// TIA Portal V17 export
// export: Created 2025-03-12T15:33:50.5234249Z, ExportSetting WithDefaults, DisplayName Totally Integrated Automation Portal, DisplayVersion V17 Update 8, DisplayName TIA Portal Openness, DisplayVersion V17 Update 8, DisplayName TIA Portal Version Control Interface, DisplayVersion V17, DisplayName SINAMICS Startdrive Advanced, DisplayVersion V17 SP2, DisplayName SINAMICS Startdrive G110M, G120, G120C, G120D, G120P, G115D, DisplayVersion V17 SP2, DisplayName SINAMICS Startdrive G130, G150, S120, S150, SINAMICS MV, S210, DisplayVersion V17 SP2, DisplayName STEP 7 Professional, DisplayVersion V17 Update 8, DisplayName SINUMERIK ONE STEP 7 Toolbox, DisplayVersion V17 Update 12, DisplayName SINUMERIK 840D sl STEP 7 Toolbox, DisplayVersion V17 Update 12, DisplayName STEP 7 Safety, DisplayVersion V17 Update 6, DisplayName WinCC Advanced, DisplayVersion V17 Update 8
FUNCTION "FC1101_MACHINE_SEQUENCE" : Void   // FC1101, LAD
{ S7_Optimized_Access := 'FALSE' }
AUTHOR : ETXETAR
VERSION : 1.0
// stored: AutoNumber false, IsIECCheckEnabled false, SetENOAutomatically false, UDAEnableTagReadback false
   VAR_TEMP
      PHD_ARM1 : Bool;   // PART HANDLING DEVICE ARM 1
      PHD_ARM2 : Bool;   // PART HANDLING DEVICE ARM 2
      QC_AUXILIARY : Bool;   // QUALITY CHECK AUXILIARY
   END_VAR
   VAR CONSTANT
      FC_NUMBER : DInt := 1101;   // FC NUMBER
   END_VAR
   VAR_TEMP   // added for the SCL form of the ladder/FBD networks
      _w1 : Bool;
      _w2 : Bool;
      _w3 : Bool;
   END_VAR
BEGIN

REGION Network 1: GENERAL CONDITIONS
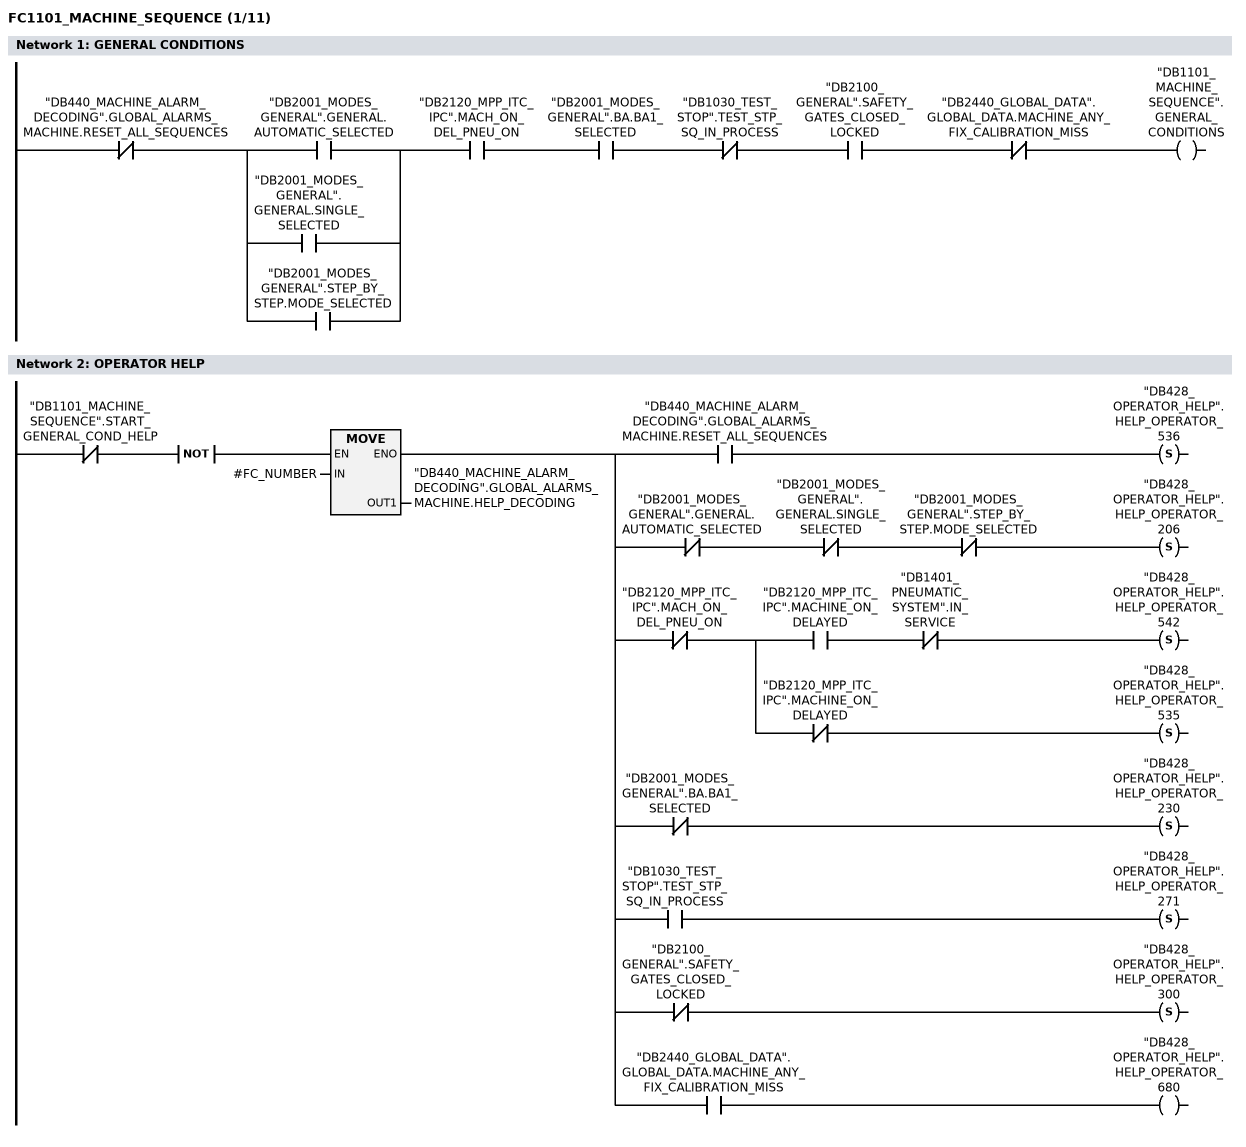
   RUNG wire#powerrail
      I_Contact( "DB440_MACHINE_ALARM_DECODING".GLOBAL_ALARMS_MACHINE.RESET_ALL_SEQUENCES )
      wire#w1
      Contact( "DB2001_MODES_GENERAL".GENERAL.AUTOMATIC_SELECTED )
      wire#w2
      Contact( "DB2120_MPP_ITC_IPC".MACH_ON_DEL_PNEU_ON )
      Contact( "DB2001_MODES_GENERAL".BA.BA1_SELECTED )
      I_Contact( "DB1030_TEST_STOP".TEST_STP_SQ_IN_PROCESS )
      Contact( "DB2100_GENERAL".SAFETY_GATES_CLOSED_LOCKED )
      I_Contact( "DB2440_GLOBAL_DATA".GLOBAL_DATA.MACHINE_ANY_FIX_CALIBRATION_MISS )
      Coil( "DB1101_MACHINE_SEQUENCE".GENERAL_CONDITIONS )
   END_RUNG
   RUNG wire#w1
      Contact( "DB2001_MODES_GENERAL".GENERAL.SINGLE_SELECTED )
   END_RUNG wire#w2
   RUNG wire#w1
      Contact( "DB2001_MODES_GENERAL".STEP_BY_STEP.MODE_SELECTED )
   END_RUNG wire#w2
   // the same network as SCL:
   "DB1101_MACHINE_SEQUENCE".GENERAL_CONDITIONS := NOT "DB440_MACHINE_ALARM_DECODING".GLOBAL_ALARMS_MACHINE.RESET_ALL_SEQUENCES AND ("DB2001_MODES_GENERAL".GENERAL.AUTOMATIC_SELECTED OR "DB2001_MODES_GENERAL".GENERAL.SINGLE_SELECTED OR "DB2001_MODES_GENERAL".STEP_BY_STEP.MODE_SELECTED) AND "DB2120_MPP_ITC_IPC".MACH_ON_DEL_PNEU_ON AND "DB2001_MODES_GENERAL".BA.BA1_SELECTED AND NOT "DB1030_TEST_STOP".TEST_STP_SQ_IN_PROCESS AND "DB2100_GENERAL".SAFETY_GATES_CLOSED_LOCKED AND NOT "DB2440_GLOBAL_DATA".GLOBAL_DATA.MACHINE_ANY_FIX_CALIBRATION_MISS;
END_REGION

REGION Network 2: OPERATOR HELP
   RUNG wire#powerrail
      I_Contact( "DB1101_MACHINE_SEQUENCE".START_GENERAL_COND_HELP )
      Not()
      { S7_GenerateENO := "TRUE" } Move(in := #FC_NUMBER, out1 => "DB440_MACHINE_ALARM_DECODING".GLOBAL_ALARMS_MACHINE.HELP_DECODING)
      wire#w1
      Contact( "DB440_MACHINE_ALARM_DECODING".GLOBAL_ALARMS_MACHINE.RESET_ALL_SEQUENCES )
      S_Coil( "DB428_OPERATOR_HELP".HELP_OPERATOR_536 )
   END_RUNG
   RUNG wire#w1
      I_Contact( "DB2001_MODES_GENERAL".GENERAL.AUTOMATIC_SELECTED )
      I_Contact( "DB2001_MODES_GENERAL".GENERAL.SINGLE_SELECTED )
      I_Contact( "DB2001_MODES_GENERAL".STEP_BY_STEP.MODE_SELECTED )
      S_Coil( "DB428_OPERATOR_HELP".HELP_OPERATOR_206 )
   END_RUNG
   RUNG wire#w1
      I_Contact( "DB2120_MPP_ITC_IPC".MACH_ON_DEL_PNEU_ON )
      wire#w2
      Contact( "DB2120_MPP_ITC_IPC".MACHINE_ON_DELAYED )
      I_Contact( "DB1401_PNEUMATIC_SYSTEM".IN_SERVICE )
      S_Coil( "DB428_OPERATOR_HELP".HELP_OPERATOR_542 )
   END_RUNG
   RUNG wire#w2
      I_Contact( "DB2120_MPP_ITC_IPC".MACHINE_ON_DELAYED )
      S_Coil( "DB428_OPERATOR_HELP".HELP_OPERATOR_535 )
   END_RUNG
   RUNG wire#w1
      I_Contact( "DB2001_MODES_GENERAL".BA.BA1_SELECTED )
      S_Coil( "DB428_OPERATOR_HELP".HELP_OPERATOR_230 )
   END_RUNG
   RUNG wire#w1
      Contact( "DB1030_TEST_STOP".TEST_STP_SQ_IN_PROCESS )
      S_Coil( "DB428_OPERATOR_HELP".HELP_OPERATOR_271 )
   END_RUNG
   RUNG wire#w1
      I_Contact( "DB2100_GENERAL".SAFETY_GATES_CLOSED_LOCKED )
      S_Coil( "DB428_OPERATOR_HELP".HELP_OPERATOR_300 )
   END_RUNG
   RUNG wire#w1
      Contact( "DB2440_GLOBAL_DATA".GLOBAL_DATA.MACHINE_ANY_FIX_CALIBRATION_MISS )
      Coil( "DB428_OPERATOR_HELP".HELP_OPERATOR_680 )
   END_RUNG
   // the same network as SCL:
   // ENO of a box is taken as its EN; it also drops when the box reports an error
   #_w1 := NOT (NOT "DB1101_MACHINE_SEQUENCE".START_GENERAL_COND_HELP);
   IF #_w1 THEN "DB440_MACHINE_ALARM_DECODING".GLOBAL_ALARMS_MACHINE.HELP_DECODING := #FC_NUMBER; END_IF;
   IF #_w1 AND "DB440_MACHINE_ALARM_DECODING".GLOBAL_ALARMS_MACHINE.RESET_ALL_SEQUENCES THEN
       "DB428_OPERATOR_HELP".HELP_OPERATOR_536 := TRUE;
   END_IF;
   IF #_w1 AND NOT "DB2001_MODES_GENERAL".GENERAL.AUTOMATIC_SELECTED AND NOT "DB2001_MODES_GENERAL".GENERAL.SINGLE_SELECTED AND NOT "DB2001_MODES_GENERAL".STEP_BY_STEP.MODE_SELECTED THEN
       "DB428_OPERATOR_HELP".HELP_OPERATOR_206 := TRUE;
   END_IF;
   #_w2 := #_w1 AND NOT "DB2120_MPP_ITC_IPC".MACH_ON_DEL_PNEU_ON;
   IF #_w2 AND "DB2120_MPP_ITC_IPC".MACHINE_ON_DELAYED AND NOT "DB1401_PNEUMATIC_SYSTEM".IN_SERVICE THEN
       "DB428_OPERATOR_HELP".HELP_OPERATOR_542 := TRUE;
   END_IF;
   IF #_w2 AND NOT "DB2120_MPP_ITC_IPC".MACHINE_ON_DELAYED THEN
       "DB428_OPERATOR_HELP".HELP_OPERATOR_535 := TRUE;
   END_IF;
   IF #_w1 AND NOT "DB2001_MODES_GENERAL".BA.BA1_SELECTED THEN
       "DB428_OPERATOR_HELP".HELP_OPERATOR_230 := TRUE;
   END_IF;
   IF #_w1 AND "DB1030_TEST_STOP".TEST_STP_SQ_IN_PROCESS THEN
       "DB428_OPERATOR_HELP".HELP_OPERATOR_271 := TRUE;
   END_IF;
   IF #_w1 AND NOT "DB2100_GENERAL".SAFETY_GATES_CLOSED_LOCKED THEN
       "DB428_OPERATOR_HELP".HELP_OPERATOR_300 := TRUE;
   END_IF;
   "DB428_OPERATOR_HELP".HELP_OPERATOR_680 := #_w1 AND "DB2440_GLOBAL_DATA".GLOBAL_DATA.MACHINE_ANY_FIX_CALIBRATION_MISS;
END_REGION

REGION Network 3: INITIAL CONDITIONS
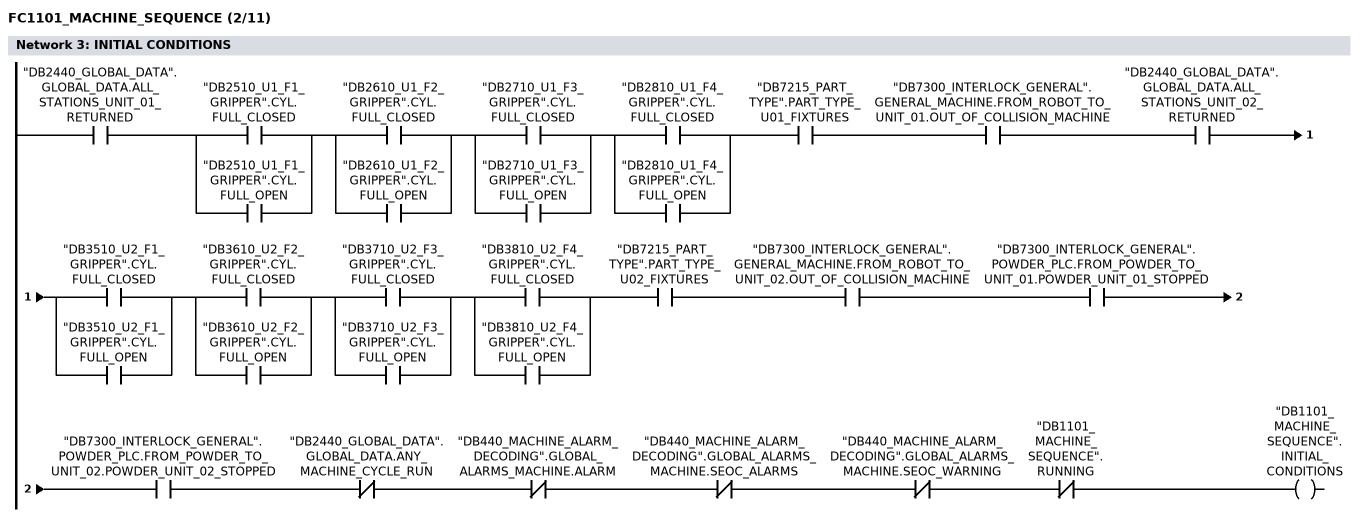
   RUNG wire#powerrail
      Contact( "DB2440_GLOBAL_DATA".GLOBAL_DATA.ALL_STATIONS_UNIT_01_RETURNED )
      wire#w1
      Contact( "DB2510_U1_F1_GRIPPER".CYL.FULL_CLOSED )
      wire#w2
      Contact( "DB2610_U1_F2_GRIPPER".CYL.FULL_CLOSED )
      wire#w3
      Contact( "DB2710_U1_F3_GRIPPER".CYL.FULL_CLOSED )
      wire#w4
      Contact( "DB2810_U1_F4_GRIPPER".CYL.FULL_CLOSED )
      wire#w5
      Contact( "DB7215_PART_TYPE".PART_TYPE_U01_FIXTURES )
      Contact( "DB7300_INTERLOCK_GENERAL".GENERAL_MACHINE.FROM_ROBOT_TO_UNIT_01.OUT_OF_COLLISION_MACHINE )
      Contact( "DB2440_GLOBAL_DATA".GLOBAL_DATA.ALL_STATIONS_UNIT_02_RETURNED )
      wire#w6
      Contact( "DB3510_U2_F1_GRIPPER".CYL.FULL_CLOSED )
      wire#w7
      Contact( "DB3610_U2_F2_GRIPPER".CYL.FULL_CLOSED )
      wire#w8
      Contact( "DB3710_U2_F3_GRIPPER".CYL.FULL_CLOSED )
      wire#w9
      Contact( "DB3810_U2_F4_GRIPPER".CYL.FULL_CLOSED )
      wire#w10
      Contact( "DB7215_PART_TYPE".PART_TYPE_U02_FIXTURES )
      Contact( "DB7300_INTERLOCK_GENERAL".GENERAL_MACHINE.FROM_ROBOT_TO_UNIT_02.OUT_OF_COLLISION_MACHINE )
      Contact( "DB7300_INTERLOCK_GENERAL".POWDER_PLC.FROM_POWDER_TO_UNIT_01.POWDER_UNIT_01_STOPPED )
      Contact( "DB7300_INTERLOCK_GENERAL".POWDER_PLC.FROM_POWDER_TO_UNIT_02.POWDER_UNIT_02_STOPPED )
      I_Contact( "DB2440_GLOBAL_DATA".GLOBAL_DATA.ANY_MACHINE_CYCLE_RUN )
      I_Contact( "DB440_MACHINE_ALARM_DECODING".GLOBAL_ALARMS_MACHINE.ALARM )
      I_Contact( "DB440_MACHINE_ALARM_DECODING".GLOBAL_ALARMS_MACHINE.SEOC_ALARMS )
      I_Contact( "DB440_MACHINE_ALARM_DECODING".GLOBAL_ALARMS_MACHINE.SEOC_WARNING )
      I_Contact( "DB1101_MACHINE_SEQUENCE".RUNNING )
      Coil( "DB1101_MACHINE_SEQUENCE".INITIAL_CONDITIONS )
   END_RUNG
   RUNG wire#w1
      Contact( "DB2510_U1_F1_GRIPPER".CYL.FULL_OPEN )
   END_RUNG wire#w2
   RUNG wire#w2
      Contact( "DB2610_U1_F2_GRIPPER".CYL.FULL_OPEN )
   END_RUNG wire#w3
   RUNG wire#w3
      Contact( "DB2710_U1_F3_GRIPPER".CYL.FULL_OPEN )
   END_RUNG wire#w4
   RUNG wire#w4
      Contact( "DB2810_U1_F4_GRIPPER".CYL.FULL_OPEN )
   END_RUNG wire#w5
   RUNG wire#w6
      Contact( "DB3510_U2_F1_GRIPPER".CYL.FULL_OPEN )
   END_RUNG wire#w7
   RUNG wire#w7
      Contact( "DB3610_U2_F2_GRIPPER".CYL.FULL_OPEN )
   END_RUNG wire#w8
   RUNG wire#w8
      Contact( "DB3710_U2_F3_GRIPPER".CYL.FULL_OPEN )
   END_RUNG wire#w9
   RUNG wire#w9
      Contact( "DB3810_U2_F4_GRIPPER".CYL.FULL_OPEN )
   END_RUNG wire#w10
   // the same network as SCL:
   "DB1101_MACHINE_SEQUENCE".INITIAL_CONDITIONS := "DB2440_GLOBAL_DATA".GLOBAL_DATA.ALL_STATIONS_UNIT_01_RETURNED AND ("DB2510_U1_F1_GRIPPER".CYL.FULL_CLOSED OR "DB2510_U1_F1_GRIPPER".CYL.FULL_OPEN) AND ("DB2610_U1_F2_GRIPPER".CYL.FULL_CLOSED OR "DB2610_U1_F2_GRIPPER".CYL.FULL_OPEN) AND ("DB2710_U1_F3_GRIPPER".CYL.FULL_CLOSED OR "DB2710_U1_F3_GRIPPER".CYL.FULL_OPEN) AND ("DB2810_U1_F4_GRIPPER".CYL.FULL_CLOSED OR "DB2810_U1_F4_GRIPPER".CYL.FULL_OPEN) AND "DB7215_PART_TYPE".PART_TYPE_U01_FIXTURES AND "DB7300_INTERLOCK_GENERAL".GENERAL_MACHINE.FROM_ROBOT_TO_UNIT_01.OUT_OF_COLLISION_MACHINE AND "DB2440_GLOBAL_DATA".GLOBAL_DATA.ALL_STATIONS_UNIT_02_RETURNED AND ("DB3510_U2_F1_GRIPPER".CYL.FULL_CLOSED OR "DB3510_U2_F1_GRIPPER".CYL.FULL_OPEN) AND ("DB3610_U2_F2_GRIPPER".CYL.FULL_CLOSED OR "DB3610_U2_F2_GRIPPER".CYL.FULL_OPEN) AND ("DB3710_U2_F3_GRIPPER".CYL.FULL_CLOSED OR "DB3710_U2_F3_GRIPPER".CYL.FULL_OPEN) AND ("DB3810_U2_F4_GRIPPER".CYL.FULL_CLOSED OR "DB3810_U2_F4_GRIPPER".CYL.FULL_OPEN) AND "DB7215_PART_TYPE".PART_TYPE_U02_FIXTURES AND "DB7300_INTERLOCK_GENERAL".GENERAL_MACHINE.FROM_ROBOT_TO_UNIT_02.OUT_OF_COLLISION_MACHINE AND "DB7300_INTERLOCK_GENERAL".POWDER_PLC.FROM_POWDER_TO_UNIT_01.POWDER_UNIT_01_STOPPED AND "DB7300_INTERLOCK_GENERAL".POWDER_PLC.FROM_POWDER_TO_UNIT_02.POWDER_UNIT_02_STOPPED AND NOT "DB2440_GLOBAL_DATA".GLOBAL_DATA.ANY_MACHINE_CYCLE_RUN AND NOT "DB440_MACHINE_ALARM_DECODING".GLOBAL_ALARMS_MACHINE.ALARM AND NOT "DB440_MACHINE_ALARM_DECODING".GLOBAL_ALARMS_MACHINE.SEOC_ALARMS AND NOT "DB440_MACHINE_ALARM_DECODING".GLOBAL_ALARMS_MACHINE.SEOC_WARNING AND NOT "DB1101_MACHINE_SEQUENCE".RUNNING;
END_REGION

REGION Network 4: OPERATOR HELP
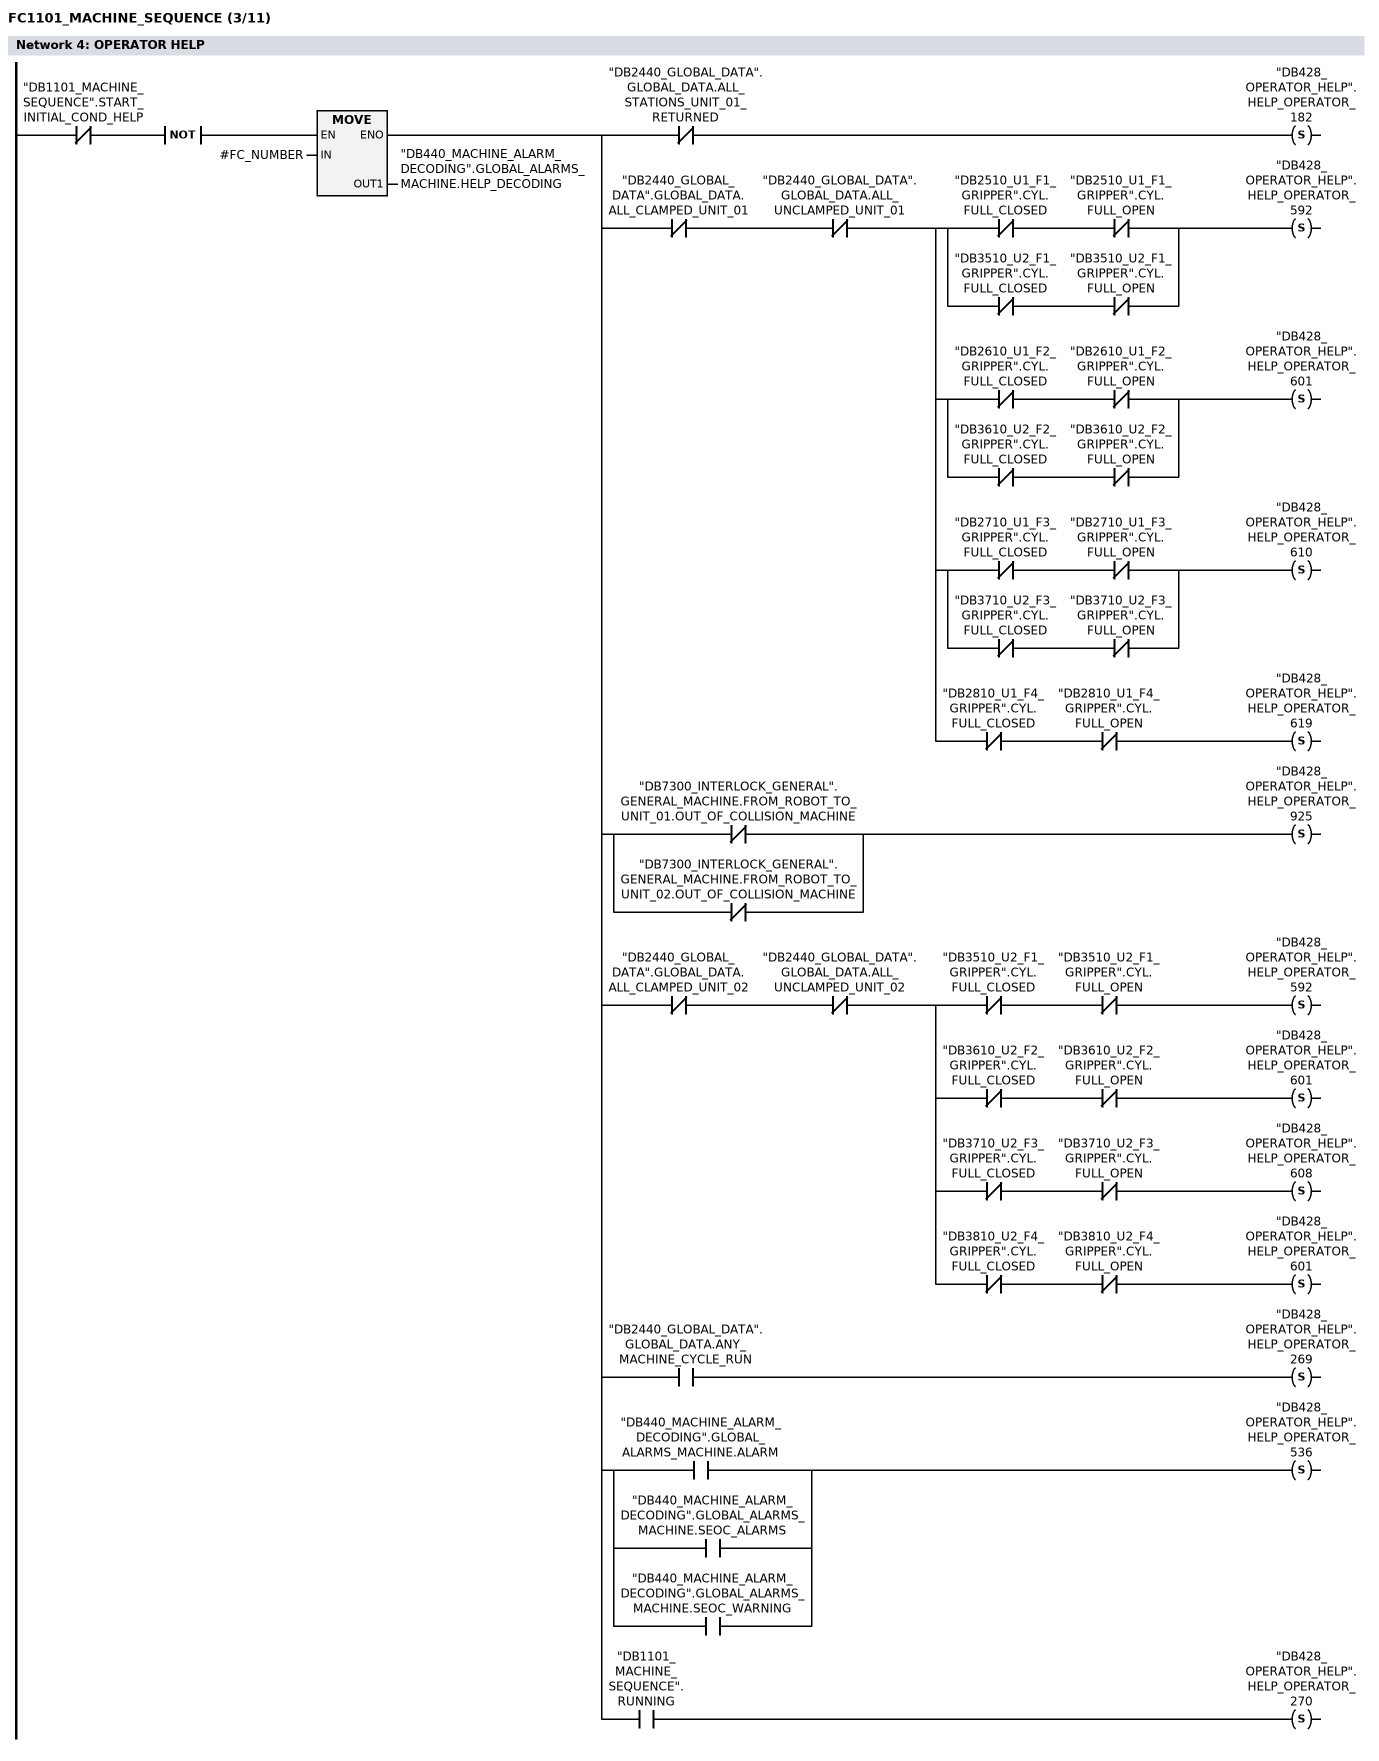
   RUNG wire#powerrail
      I_Contact( "DB1101_MACHINE_SEQUENCE".START_INITIAL_COND_HELP )
      Not()
      { S7_GenerateENO := "TRUE" } Move(in := #FC_NUMBER, out1 => "DB440_MACHINE_ALARM_DECODING".GLOBAL_ALARMS_MACHINE.HELP_DECODING)
      wire#w1
      I_Contact( "DB2440_GLOBAL_DATA".GLOBAL_DATA.ALL_STATIONS_UNIT_01_RETURNED )
      S_Coil( "DB428_OPERATOR_HELP".HELP_OPERATOR_182 )
   END_RUNG
   RUNG wire#w1
      I_Contact( "DB2440_GLOBAL_DATA".GLOBAL_DATA.ALL_CLAMPED_UNIT_01 )
      I_Contact( "DB2440_GLOBAL_DATA".GLOBAL_DATA.ALL_UNCLAMPED_UNIT_01 )
      wire#w2
      I_Contact( "DB2510_U1_F1_GRIPPER".CYL.FULL_CLOSED )
      I_Contact( "DB2510_U1_F1_GRIPPER".CYL.FULL_OPEN )
      wire#w3
      S_Coil( "DB428_OPERATOR_HELP".HELP_OPERATOR_592 )
   END_RUNG
   RUNG wire#w2
      I_Contact( "DB3510_U2_F1_GRIPPER".CYL.FULL_CLOSED )
      I_Contact( "DB3510_U2_F1_GRIPPER".CYL.FULL_OPEN )
   END_RUNG wire#w3
   RUNG wire#w2
      I_Contact( "DB2610_U1_F2_GRIPPER".CYL.FULL_CLOSED )
      I_Contact( "DB2610_U1_F2_GRIPPER".CYL.FULL_OPEN )
      wire#w4
      S_Coil( "DB428_OPERATOR_HELP".HELP_OPERATOR_601 )
   END_RUNG
   RUNG wire#w2
      I_Contact( "DB3610_U2_F2_GRIPPER".CYL.FULL_CLOSED )
      I_Contact( "DB3610_U2_F2_GRIPPER".CYL.FULL_OPEN )
   END_RUNG wire#w4
   RUNG wire#w2
      I_Contact( "DB2710_U1_F3_GRIPPER".CYL.FULL_CLOSED )
      I_Contact( "DB2710_U1_F3_GRIPPER".CYL.FULL_OPEN )
      wire#w5
      S_Coil( "DB428_OPERATOR_HELP".HELP_OPERATOR_610 )
   END_RUNG
   RUNG wire#w2
      I_Contact( "DB3710_U2_F3_GRIPPER".CYL.FULL_CLOSED )
      I_Contact( "DB3710_U2_F3_GRIPPER".CYL.FULL_OPEN )
   END_RUNG wire#w5
   RUNG wire#w2
      I_Contact( "DB2810_U1_F4_GRIPPER".CYL.FULL_CLOSED )
      I_Contact( "DB2810_U1_F4_GRIPPER".CYL.FULL_OPEN )
      S_Coil( "DB428_OPERATOR_HELP".HELP_OPERATOR_619 )
   END_RUNG
   RUNG wire#w1
      I_Contact( "DB7300_INTERLOCK_GENERAL".GENERAL_MACHINE.FROM_ROBOT_TO_UNIT_01.OUT_OF_COLLISION_MACHINE )
      wire#w6
      S_Coil( "DB428_OPERATOR_HELP".HELP_OPERATOR_925 )
   END_RUNG
   RUNG wire#w1
      I_Contact( "DB7300_INTERLOCK_GENERAL".GENERAL_MACHINE.FROM_ROBOT_TO_UNIT_02.OUT_OF_COLLISION_MACHINE )
   END_RUNG wire#w6
   RUNG wire#w1
      I_Contact( "DB2440_GLOBAL_DATA".GLOBAL_DATA.ALL_CLAMPED_UNIT_02 )
      I_Contact( "DB2440_GLOBAL_DATA".GLOBAL_DATA.ALL_UNCLAMPED_UNIT_02 )
      wire#w7
      I_Contact( "DB3510_U2_F1_GRIPPER".CYL.FULL_CLOSED )
      I_Contact( "DB3510_U2_F1_GRIPPER".CYL.FULL_OPEN )
      S_Coil( "DB428_OPERATOR_HELP".HELP_OPERATOR_592 )
   END_RUNG
   RUNG wire#w7
      I_Contact( "DB3610_U2_F2_GRIPPER".CYL.FULL_CLOSED )
      I_Contact( "DB3610_U2_F2_GRIPPER".CYL.FULL_OPEN )
      S_Coil( "DB428_OPERATOR_HELP".HELP_OPERATOR_601 )
   END_RUNG
   RUNG wire#w7
      I_Contact( "DB3710_U2_F3_GRIPPER".CYL.FULL_CLOSED )
      I_Contact( "DB3710_U2_F3_GRIPPER".CYL.FULL_OPEN )
      S_Coil( "DB428_OPERATOR_HELP".HELP_OPERATOR_608 )
   END_RUNG
   RUNG wire#w7
      I_Contact( "DB3810_U2_F4_GRIPPER".CYL.FULL_CLOSED )
      I_Contact( "DB3810_U2_F4_GRIPPER".CYL.FULL_OPEN )
      S_Coil( "DB428_OPERATOR_HELP".HELP_OPERATOR_601 )
   END_RUNG
   RUNG wire#w1
      Contact( "DB2440_GLOBAL_DATA".GLOBAL_DATA.ANY_MACHINE_CYCLE_RUN )
      S_Coil( "DB428_OPERATOR_HELP".HELP_OPERATOR_269 )
   END_RUNG
   RUNG wire#w1
      Contact( "DB440_MACHINE_ALARM_DECODING".GLOBAL_ALARMS_MACHINE.ALARM )
      wire#w8
      S_Coil( "DB428_OPERATOR_HELP".HELP_OPERATOR_536 )
   END_RUNG
   RUNG wire#w1
      Contact( "DB440_MACHINE_ALARM_DECODING".GLOBAL_ALARMS_MACHINE.SEOC_ALARMS )
   END_RUNG wire#w8
   RUNG wire#w1
      Contact( "DB440_MACHINE_ALARM_DECODING".GLOBAL_ALARMS_MACHINE.SEOC_WARNING )
   END_RUNG wire#w8
   RUNG wire#w1
      Contact( "DB1101_MACHINE_SEQUENCE".RUNNING )
      S_Coil( "DB428_OPERATOR_HELP".HELP_OPERATOR_270 )
   END_RUNG
   // the same network as SCL:
   // ENO of a box is taken as its EN; it also drops when the box reports an error
   #_w1 := NOT (NOT "DB1101_MACHINE_SEQUENCE".START_INITIAL_COND_HELP);
   IF #_w1 THEN "DB440_MACHINE_ALARM_DECODING".GLOBAL_ALARMS_MACHINE.HELP_DECODING := #FC_NUMBER; END_IF;
   IF #_w1 AND NOT "DB2440_GLOBAL_DATA".GLOBAL_DATA.ALL_STATIONS_UNIT_01_RETURNED THEN
       "DB428_OPERATOR_HELP".HELP_OPERATOR_182 := TRUE;
   END_IF;
   #_w2 := #_w1 AND NOT "DB2440_GLOBAL_DATA".GLOBAL_DATA.ALL_CLAMPED_UNIT_01 AND NOT "DB2440_GLOBAL_DATA".GLOBAL_DATA.ALL_UNCLAMPED_UNIT_01;
   IF #_w2 AND ((NOT "DB2510_U1_F1_GRIPPER".CYL.FULL_CLOSED AND NOT "DB2510_U1_F1_GRIPPER".CYL.FULL_OPEN) OR (NOT "DB3510_U2_F1_GRIPPER".CYL.FULL_CLOSED AND NOT "DB3510_U2_F1_GRIPPER".CYL.FULL_OPEN)) THEN
       "DB428_OPERATOR_HELP".HELP_OPERATOR_592 := TRUE;
   END_IF;
   IF #_w2 AND ((NOT "DB2610_U1_F2_GRIPPER".CYL.FULL_CLOSED AND NOT "DB2610_U1_F2_GRIPPER".CYL.FULL_OPEN) OR (NOT "DB3610_U2_F2_GRIPPER".CYL.FULL_CLOSED AND NOT "DB3610_U2_F2_GRIPPER".CYL.FULL_OPEN)) THEN
       "DB428_OPERATOR_HELP".HELP_OPERATOR_601 := TRUE;
   END_IF;
   IF #_w2 AND ((NOT "DB2710_U1_F3_GRIPPER".CYL.FULL_CLOSED AND NOT "DB2710_U1_F3_GRIPPER".CYL.FULL_OPEN) OR (NOT "DB3710_U2_F3_GRIPPER".CYL.FULL_CLOSED AND NOT "DB3710_U2_F3_GRIPPER".CYL.FULL_OPEN)) THEN
       "DB428_OPERATOR_HELP".HELP_OPERATOR_610 := TRUE;
   END_IF;
   IF #_w2 AND NOT "DB2810_U1_F4_GRIPPER".CYL.FULL_CLOSED AND NOT "DB2810_U1_F4_GRIPPER".CYL.FULL_OPEN THEN
       "DB428_OPERATOR_HELP".HELP_OPERATOR_619 := TRUE;
   END_IF;
   IF #_w1 AND (NOT "DB7300_INTERLOCK_GENERAL".GENERAL_MACHINE.FROM_ROBOT_TO_UNIT_01.OUT_OF_COLLISION_MACHINE OR NOT "DB7300_INTERLOCK_GENERAL".GENERAL_MACHINE.FROM_ROBOT_TO_UNIT_02.OUT_OF_COLLISION_MACHINE) THEN
       "DB428_OPERATOR_HELP".HELP_OPERATOR_925 := TRUE;
   END_IF;
   #_w3 := #_w1 AND NOT "DB2440_GLOBAL_DATA".GLOBAL_DATA.ALL_CLAMPED_UNIT_02 AND NOT "DB2440_GLOBAL_DATA".GLOBAL_DATA.ALL_UNCLAMPED_UNIT_02;
   IF #_w3 AND NOT "DB3510_U2_F1_GRIPPER".CYL.FULL_CLOSED AND NOT "DB3510_U2_F1_GRIPPER".CYL.FULL_OPEN THEN
       "DB428_OPERATOR_HELP".HELP_OPERATOR_592 := TRUE;
   END_IF;
   IF #_w3 AND NOT "DB3610_U2_F2_GRIPPER".CYL.FULL_CLOSED AND NOT "DB3610_U2_F2_GRIPPER".CYL.FULL_OPEN THEN
       "DB428_OPERATOR_HELP".HELP_OPERATOR_601 := TRUE;
   END_IF;
   IF #_w3 AND NOT "DB3710_U2_F3_GRIPPER".CYL.FULL_CLOSED AND NOT "DB3710_U2_F3_GRIPPER".CYL.FULL_OPEN THEN
       "DB428_OPERATOR_HELP".HELP_OPERATOR_608 := TRUE;
   END_IF;
   IF #_w3 AND NOT "DB3810_U2_F4_GRIPPER".CYL.FULL_CLOSED AND NOT "DB3810_U2_F4_GRIPPER".CYL.FULL_OPEN THEN
       "DB428_OPERATOR_HELP".HELP_OPERATOR_601 := TRUE;
   END_IF;
   IF #_w1 AND "DB2440_GLOBAL_DATA".GLOBAL_DATA.ANY_MACHINE_CYCLE_RUN THEN
       "DB428_OPERATOR_HELP".HELP_OPERATOR_269 := TRUE;
   END_IF;
   IF #_w1 AND ("DB440_MACHINE_ALARM_DECODING".GLOBAL_ALARMS_MACHINE.ALARM OR "DB440_MACHINE_ALARM_DECODING".GLOBAL_ALARMS_MACHINE.SEOC_ALARMS OR "DB440_MACHINE_ALARM_DECODING".GLOBAL_ALARMS_MACHINE.SEOC_WARNING) THEN
       "DB428_OPERATOR_HELP".HELP_OPERATOR_536 := TRUE;
   END_IF;
   IF #_w1 AND "DB1101_MACHINE_SEQUENCE".RUNNING THEN
       "DB428_OPERATOR_HELP".HELP_OPERATOR_270 := TRUE;
   END_IF;
END_REGION

REGION Network 5: START REQUEST
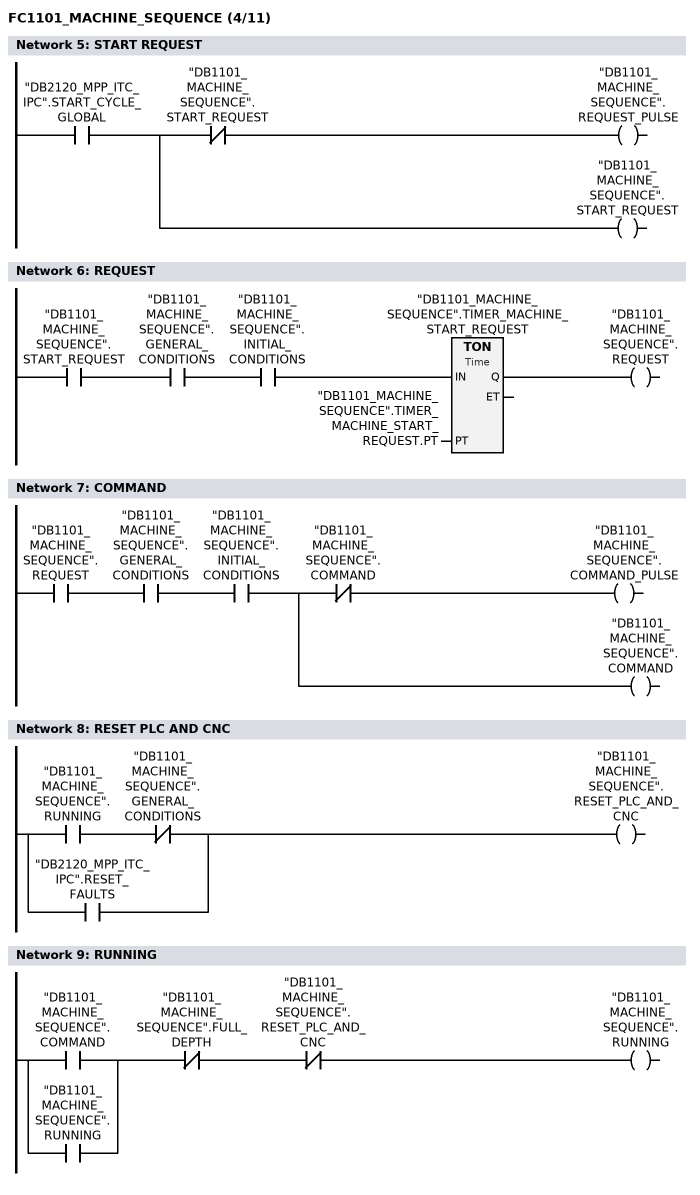
   RUNG wire#powerrail
      Contact( "DB2120_MPP_ITC_IPC".START_CYCLE_GLOBAL )
      wire#w1
      I_Contact( "DB1101_MACHINE_SEQUENCE".START_REQUEST )
      Coil( "DB1101_MACHINE_SEQUENCE".REQUEST_PULSE )
   END_RUNG
   RUNG wire#w1
      Coil( "DB1101_MACHINE_SEQUENCE".START_REQUEST )
   END_RUNG
   // the same network as SCL:
   "DB1101_MACHINE_SEQUENCE".REQUEST_PULSE := "DB2120_MPP_ITC_IPC".START_CYCLE_GLOBAL AND NOT "DB1101_MACHINE_SEQUENCE".START_REQUEST;
   "DB1101_MACHINE_SEQUENCE".START_REQUEST := "DB2120_MPP_ITC_IPC".START_CYCLE_GLOBAL;
END_REGION

REGION Network 6: REQUEST
   RUNG wire#powerrail
      Contact( "DB1101_MACHINE_SEQUENCE".START_REQUEST )
      Contact( "DB1101_MACHINE_SEQUENCE".GENERAL_CONDITIONS )
      Contact( "DB1101_MACHINE_SEQUENCE".INITIAL_CONDITIONS )
      { S7_Templates := "time_type := Time" } "DB1101_MACHINE_SEQUENCE".TIMER_MACHINE_START_REQUEST.TON(pt := "DB1101_MACHINE_SEQUENCE".TIMER_MACHINE_START_REQUEST.PT, et =>)
      Coil( "DB1101_MACHINE_SEQUENCE".REQUEST )
   END_RUNG
   // the same network as SCL:
   "DB1101_MACHINE_SEQUENCE".TIMER_MACHINE_START_REQUEST.TON(IN := "DB1101_MACHINE_SEQUENCE".START_REQUEST AND "DB1101_MACHINE_SEQUENCE".GENERAL_CONDITIONS AND "DB1101_MACHINE_SEQUENCE".INITIAL_CONDITIONS,
                           PT := "DB1101_MACHINE_SEQUENCE".TIMER_MACHINE_START_REQUEST.PT);
   "DB1101_MACHINE_SEQUENCE".REQUEST := "DB1101_MACHINE_SEQUENCE".TIMER_MACHINE_START_REQUEST.Q;
END_REGION

REGION Network 7: COMMAND
   RUNG wire#powerrail
      Contact( "DB1101_MACHINE_SEQUENCE".REQUEST )
      Contact( "DB1101_MACHINE_SEQUENCE".GENERAL_CONDITIONS )
      Contact( "DB1101_MACHINE_SEQUENCE".INITIAL_CONDITIONS )
      wire#w1
      I_Contact( "DB1101_MACHINE_SEQUENCE".COMMAND )
      Coil( "DB1101_MACHINE_SEQUENCE".COMMAND_PULSE )
   END_RUNG
   RUNG wire#w1
      Coil( "DB1101_MACHINE_SEQUENCE".COMMAND )
   END_RUNG
   // the same network as SCL:
   #_w1 := "DB1101_MACHINE_SEQUENCE".REQUEST AND "DB1101_MACHINE_SEQUENCE".GENERAL_CONDITIONS AND "DB1101_MACHINE_SEQUENCE".INITIAL_CONDITIONS;
   "DB1101_MACHINE_SEQUENCE".COMMAND_PULSE := #_w1 AND NOT "DB1101_MACHINE_SEQUENCE".COMMAND;
   "DB1101_MACHINE_SEQUENCE".COMMAND := #_w1;
END_REGION

REGION Network 8: RESET PLC AND CNC
   RUNG wire#powerrail
      Contact( "DB1101_MACHINE_SEQUENCE".RUNNING )
      I_Contact( "DB1101_MACHINE_SEQUENCE".GENERAL_CONDITIONS )
      wire#w1
      Coil( "DB1101_MACHINE_SEQUENCE".RESET_PLC_AND_CNC )
   END_RUNG
   RUNG wire#powerrail
      Contact( "DB2120_MPP_ITC_IPC".RESET_FAULTS )
   END_RUNG wire#w1
   // the same network as SCL:
   "DB1101_MACHINE_SEQUENCE".RESET_PLC_AND_CNC := ("DB1101_MACHINE_SEQUENCE".RUNNING AND NOT "DB1101_MACHINE_SEQUENCE".GENERAL_CONDITIONS) OR "DB2120_MPP_ITC_IPC".RESET_FAULTS;
END_REGION

REGION Network 9: RUNNING
   RUNG wire#powerrail
      Contact( "DB1101_MACHINE_SEQUENCE".COMMAND )
      wire#w1
      I_Contact( "DB1101_MACHINE_SEQUENCE".FULL_DEPTH )
      I_Contact( "DB1101_MACHINE_SEQUENCE".RESET_PLC_AND_CNC )
      Coil( "DB1101_MACHINE_SEQUENCE".RUNNING )
   END_RUNG
   RUNG wire#powerrail
      Contact( "DB1101_MACHINE_SEQUENCE".RUNNING )
   END_RUNG wire#w1
   // the same network as SCL:
   "DB1101_MACHINE_SEQUENCE".RUNNING := ("DB1101_MACHINE_SEQUENCE".COMMAND OR "DB1101_MACHINE_SEQUENCE".RUNNING) AND NOT "DB1101_MACHINE_SEQUENCE".FULL_DEPTH AND NOT "DB1101_MACHINE_SEQUENCE".RESET_PLC_AND_CNC;
END_REGION

REGION Network 10: MACHINE NO PART AT FEED UNIT 01
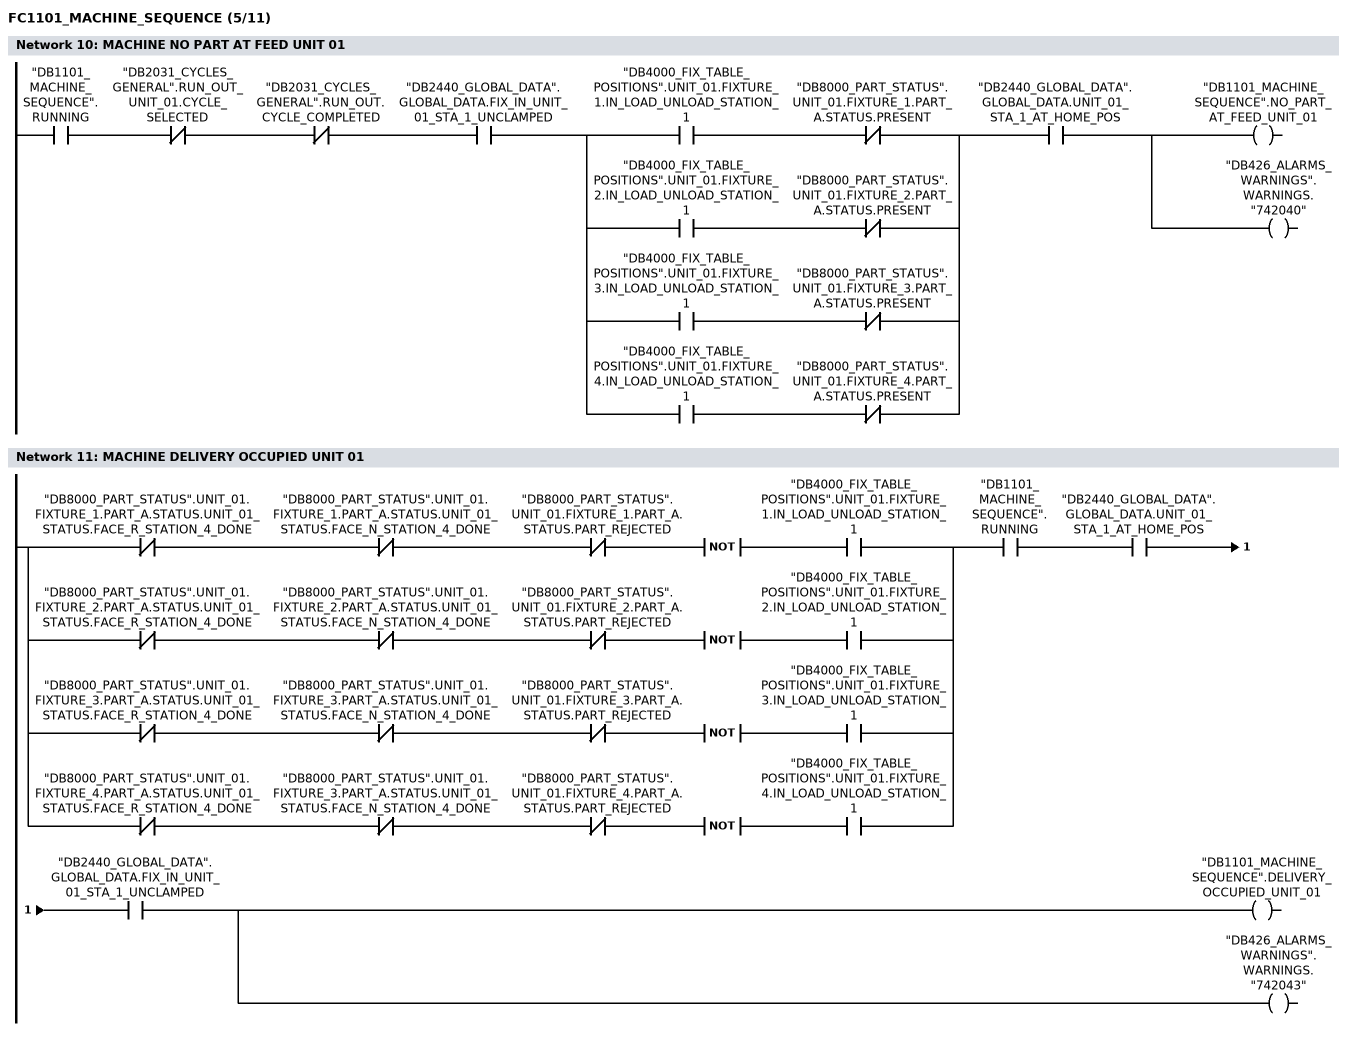
   RUNG wire#powerrail
      Contact( "DB1101_MACHINE_SEQUENCE".RUNNING )
      I_Contact( "DB2031_CYCLES_GENERAL".RUN_OUT_UNIT_01.CYCLE_SELECTED )
      I_Contact( "DB2031_CYCLES_GENERAL".RUN_OUT.CYCLE_COMPLETED )
      Contact( "DB2440_GLOBAL_DATA".GLOBAL_DATA.FIX_IN_UNIT_01_STA_1_UNCLAMPED )
      wire#w1
      Contact( "DB4000_FIX_TABLE_POSITIONS".UNIT_01.FIXTURE_1.IN_LOAD_UNLOAD_STATION_1 )
      I_Contact( "DB8000_PART_STATUS".UNIT_01.FIXTURE_1.PART_A.STATUS.PRESENT )
      wire#w2
      Contact( "DB2440_GLOBAL_DATA".GLOBAL_DATA.UNIT_01_STA_1_AT_HOME_POS )
      wire#w3
      Coil( "DB1101_MACHINE_SEQUENCE".NO_PART_AT_FEED_UNIT_01 )
   END_RUNG
   RUNG wire#w1
      Contact( "DB4000_FIX_TABLE_POSITIONS".UNIT_01.FIXTURE_2.IN_LOAD_UNLOAD_STATION_1 )
      I_Contact( "DB8000_PART_STATUS".UNIT_01.FIXTURE_2.PART_A.STATUS.PRESENT )
   END_RUNG wire#w2
   RUNG wire#w1
      Contact( "DB4000_FIX_TABLE_POSITIONS".UNIT_01.FIXTURE_3.IN_LOAD_UNLOAD_STATION_1 )
      I_Contact( "DB8000_PART_STATUS".UNIT_01.FIXTURE_3.PART_A.STATUS.PRESENT )
   END_RUNG wire#w2
   RUNG wire#w1
      Contact( "DB4000_FIX_TABLE_POSITIONS".UNIT_01.FIXTURE_4.IN_LOAD_UNLOAD_STATION_1 )
      I_Contact( "DB8000_PART_STATUS".UNIT_01.FIXTURE_4.PART_A.STATUS.PRESENT )
   END_RUNG wire#w2
   RUNG wire#w3
      Coil( "DB426_ALARMS_WARNINGS".WARNINGS."742040" )
   END_RUNG
   // the same network as SCL:
   "DB1101_MACHINE_SEQUENCE".NO_PART_AT_FEED_UNIT_01 := "DB1101_MACHINE_SEQUENCE".RUNNING AND NOT "DB2031_CYCLES_GENERAL".RUN_OUT_UNIT_01.CYCLE_SELECTED AND NOT "DB2031_CYCLES_GENERAL".RUN_OUT.CYCLE_COMPLETED AND "DB2440_GLOBAL_DATA".GLOBAL_DATA.FIX_IN_UNIT_01_STA_1_UNCLAMPED AND (("DB4000_FIX_TABLE_POSITIONS".UNIT_01.FIXTURE_1.IN_LOAD_UNLOAD_STATION_1 AND NOT "DB8000_PART_STATUS".UNIT_01.FIXTURE_1.PART_A.STATUS.PRESENT) OR ("DB4000_FIX_TABLE_POSITIONS".UNIT_01.FIXTURE_2.IN_LOAD_UNLOAD_STATION_1 AND NOT "DB8000_PART_STATUS".UNIT_01.FIXTURE_2.PART_A.STATUS.PRESENT) OR ("DB4000_FIX_TABLE_POSITIONS".UNIT_01.FIXTURE_3.IN_LOAD_UNLOAD_STATION_1 AND NOT "DB8000_PART_STATUS".UNIT_01.FIXTURE_3.PART_A.STATUS.PRESENT) OR ("DB4000_FIX_TABLE_POSITIONS".UNIT_01.FIXTURE_4.IN_LOAD_UNLOAD_STATION_1 AND NOT "DB8000_PART_STATUS".UNIT_01.FIXTURE_4.PART_A.STATUS.PRESENT)) AND "DB2440_GLOBAL_DATA".GLOBAL_DATA.UNIT_01_STA_1_AT_HOME_POS;
   "DB426_ALARMS_WARNINGS".WARNINGS."742040" := "DB1101_MACHINE_SEQUENCE".NO_PART_AT_FEED_UNIT_01;
END_REGION

REGION Network 11: MACHINE DELIVERY OCCUPIED UNIT 01
   RUNG wire#powerrail
      I_Contact( "DB8000_PART_STATUS".UNIT_01.FIXTURE_1.PART_A.STATUS.UNIT_01_STATUS.FACE_R_STATION_4_DONE )
      I_Contact( "DB8000_PART_STATUS".UNIT_01.FIXTURE_1.PART_A.STATUS.UNIT_01_STATUS.FACE_N_STATION_4_DONE )
      I_Contact( "DB8000_PART_STATUS".UNIT_01.FIXTURE_1.PART_A.STATUS.PART_REJECTED )
      Not()
      Contact( "DB4000_FIX_TABLE_POSITIONS".UNIT_01.FIXTURE_1.IN_LOAD_UNLOAD_STATION_1 )
      wire#w1
      Contact( "DB1101_MACHINE_SEQUENCE".RUNNING )
      Contact( "DB2440_GLOBAL_DATA".GLOBAL_DATA.UNIT_01_STA_1_AT_HOME_POS )
      Contact( "DB2440_GLOBAL_DATA".GLOBAL_DATA.FIX_IN_UNIT_01_STA_1_UNCLAMPED )
      wire#w2
      Coil( "DB1101_MACHINE_SEQUENCE".DELIVERY_OCCUPIED_UNIT_01 )
   END_RUNG
   RUNG wire#powerrail
      I_Contact( "DB8000_PART_STATUS".UNIT_01.FIXTURE_2.PART_A.STATUS.UNIT_01_STATUS.FACE_R_STATION_4_DONE )
      I_Contact( "DB8000_PART_STATUS".UNIT_01.FIXTURE_2.PART_A.STATUS.UNIT_01_STATUS.FACE_N_STATION_4_DONE )
      I_Contact( "DB8000_PART_STATUS".UNIT_01.FIXTURE_2.PART_A.STATUS.PART_REJECTED )
      Not()
      Contact( "DB4000_FIX_TABLE_POSITIONS".UNIT_01.FIXTURE_2.IN_LOAD_UNLOAD_STATION_1 )
   END_RUNG wire#w1
   RUNG wire#powerrail
      I_Contact( "DB8000_PART_STATUS".UNIT_01.FIXTURE_3.PART_A.STATUS.UNIT_01_STATUS.FACE_R_STATION_4_DONE )
      I_Contact( "DB8000_PART_STATUS".UNIT_01.FIXTURE_3.PART_A.STATUS.UNIT_01_STATUS.FACE_N_STATION_4_DONE )
      I_Contact( "DB8000_PART_STATUS".UNIT_01.FIXTURE_3.PART_A.STATUS.PART_REJECTED )
      Not()
      Contact( "DB4000_FIX_TABLE_POSITIONS".UNIT_01.FIXTURE_3.IN_LOAD_UNLOAD_STATION_1 )
   END_RUNG wire#w1
   RUNG wire#powerrail
      I_Contact( "DB8000_PART_STATUS".UNIT_01.FIXTURE_4.PART_A.STATUS.UNIT_01_STATUS.FACE_R_STATION_4_DONE )
      I_Contact( "DB8000_PART_STATUS".UNIT_01.FIXTURE_3.PART_A.STATUS.UNIT_01_STATUS.FACE_N_STATION_4_DONE )
      I_Contact( "DB8000_PART_STATUS".UNIT_01.FIXTURE_4.PART_A.STATUS.PART_REJECTED )
      Not()
      Contact( "DB4000_FIX_TABLE_POSITIONS".UNIT_01.FIXTURE_4.IN_LOAD_UNLOAD_STATION_1 )
   END_RUNG wire#w1
   RUNG wire#w2
      Coil( "DB426_ALARMS_WARNINGS".WARNINGS."742043" )
   END_RUNG
   // the same network as SCL:
   "DB1101_MACHINE_SEQUENCE".DELIVERY_OCCUPIED_UNIT_01 := ((NOT (NOT "DB8000_PART_STATUS".UNIT_01.FIXTURE_1.PART_A.STATUS.UNIT_01_STATUS.FACE_R_STATION_4_DONE AND NOT "DB8000_PART_STATUS".UNIT_01.FIXTURE_1.PART_A.STATUS.UNIT_01_STATUS.FACE_N_STATION_4_DONE AND NOT "DB8000_PART_STATUS".UNIT_01.FIXTURE_1.PART_A.STATUS.PART_REJECTED) AND "DB4000_FIX_TABLE_POSITIONS".UNIT_01.FIXTURE_1.IN_LOAD_UNLOAD_STATION_1) OR (NOT (NOT "DB8000_PART_STATUS".UNIT_01.FIXTURE_2.PART_A.STATUS.UNIT_01_STATUS.FACE_R_STATION_4_DONE AND NOT "DB8000_PART_STATUS".UNIT_01.FIXTURE_2.PART_A.STATUS.UNIT_01_STATUS.FACE_N_STATION_4_DONE AND NOT "DB8000_PART_STATUS".UNIT_01.FIXTURE_2.PART_A.STATUS.PART_REJECTED) AND "DB4000_FIX_TABLE_POSITIONS".UNIT_01.FIXTURE_2.IN_LOAD_UNLOAD_STATION_1) OR (NOT (NOT "DB8000_PART_STATUS".UNIT_01.FIXTURE_3.PART_A.STATUS.UNIT_01_STATUS.FACE_R_STATION_4_DONE AND NOT "DB8000_PART_STATUS".UNIT_01.FIXTURE_3.PART_A.STATUS.UNIT_01_STATUS.FACE_N_STATION_4_DONE AND NOT "DB8000_PART_STATUS".UNIT_01.FIXTURE_3.PART_A.STATUS.PART_REJECTED) AND "DB4000_FIX_TABLE_POSITIONS".UNIT_01.FIXTURE_3.IN_LOAD_UNLOAD_STATION_1) OR (NOT (NOT "DB8000_PART_STATUS".UNIT_01.FIXTURE_4.PART_A.STATUS.UNIT_01_STATUS.FACE_R_STATION_4_DONE AND NOT "DB8000_PART_STATUS".UNIT_01.FIXTURE_3.PART_A.STATUS.UNIT_01_STATUS.FACE_N_STATION_4_DONE AND NOT "DB8000_PART_STATUS".UNIT_01.FIXTURE_4.PART_A.STATUS.PART_REJECTED) AND "DB4000_FIX_TABLE_POSITIONS".UNIT_01.FIXTURE_4.IN_LOAD_UNLOAD_STATION_1)) AND "DB1101_MACHINE_SEQUENCE".RUNNING AND "DB2440_GLOBAL_DATA".GLOBAL_DATA.UNIT_01_STA_1_AT_HOME_POS AND "DB2440_GLOBAL_DATA".GLOBAL_DATA.FIX_IN_UNIT_01_STA_1_UNCLAMPED;
   "DB426_ALARMS_WARNINGS".WARNINGS."742043" := "DB1101_MACHINE_SEQUENCE".DELIVERY_OCCUPIED_UNIT_01;
END_REGION

REGION Network 12: MACHINE NO PART AT FEED UNIT 02
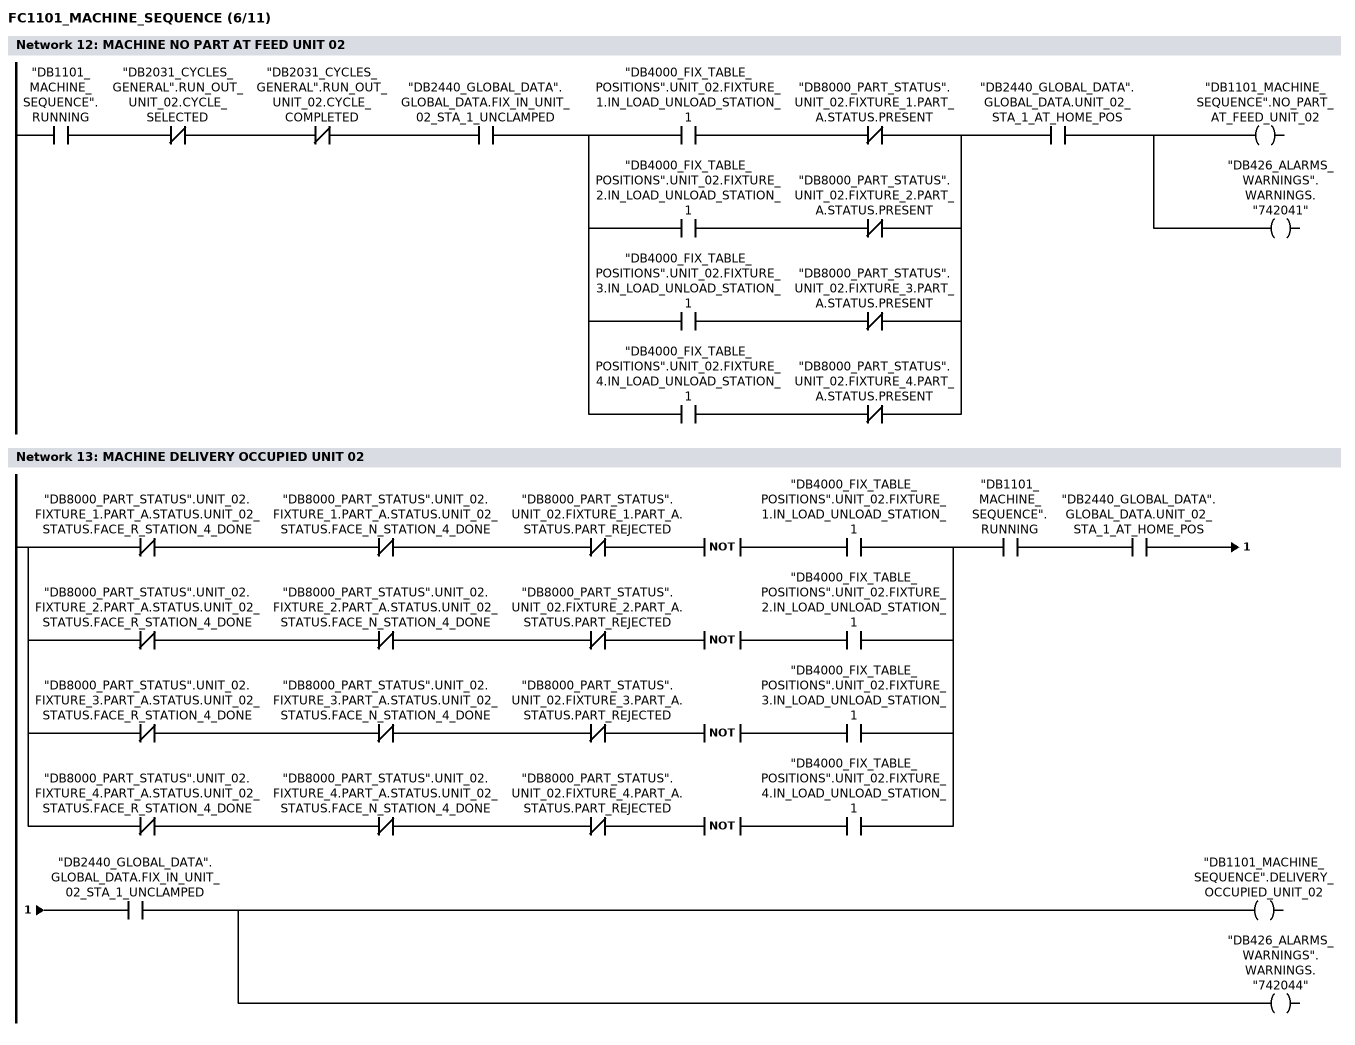
   RUNG wire#powerrail
      Contact( "DB1101_MACHINE_SEQUENCE".RUNNING )
      I_Contact( "DB2031_CYCLES_GENERAL".RUN_OUT_UNIT_02.CYCLE_SELECTED )
      I_Contact( "DB2031_CYCLES_GENERAL".RUN_OUT_UNIT_02.CYCLE_COMPLETED )
      Contact( "DB2440_GLOBAL_DATA".GLOBAL_DATA.FIX_IN_UNIT_02_STA_1_UNCLAMPED )
      wire#w1
      Contact( "DB4000_FIX_TABLE_POSITIONS".UNIT_02.FIXTURE_1.IN_LOAD_UNLOAD_STATION_1 )
      I_Contact( "DB8000_PART_STATUS".UNIT_02.FIXTURE_1.PART_A.STATUS.PRESENT )
      wire#w2
      Contact( "DB2440_GLOBAL_DATA".GLOBAL_DATA.UNIT_02_STA_1_AT_HOME_POS )
      wire#w3
      Coil( "DB1101_MACHINE_SEQUENCE".NO_PART_AT_FEED_UNIT_02 )
   END_RUNG
   RUNG wire#w1
      Contact( "DB4000_FIX_TABLE_POSITIONS".UNIT_02.FIXTURE_2.IN_LOAD_UNLOAD_STATION_1 )
      I_Contact( "DB8000_PART_STATUS".UNIT_02.FIXTURE_2.PART_A.STATUS.PRESENT )
   END_RUNG wire#w2
   RUNG wire#w1
      Contact( "DB4000_FIX_TABLE_POSITIONS".UNIT_02.FIXTURE_3.IN_LOAD_UNLOAD_STATION_1 )
      I_Contact( "DB8000_PART_STATUS".UNIT_02.FIXTURE_3.PART_A.STATUS.PRESENT )
   END_RUNG wire#w2
   RUNG wire#w1
      Contact( "DB4000_FIX_TABLE_POSITIONS".UNIT_02.FIXTURE_4.IN_LOAD_UNLOAD_STATION_1 )
      I_Contact( "DB8000_PART_STATUS".UNIT_02.FIXTURE_4.PART_A.STATUS.PRESENT )
   END_RUNG wire#w2
   RUNG wire#w3
      Coil( "DB426_ALARMS_WARNINGS".WARNINGS."742041" )
   END_RUNG
   // the same network as SCL:
   "DB1101_MACHINE_SEQUENCE".NO_PART_AT_FEED_UNIT_02 := "DB1101_MACHINE_SEQUENCE".RUNNING AND NOT "DB2031_CYCLES_GENERAL".RUN_OUT_UNIT_02.CYCLE_SELECTED AND NOT "DB2031_CYCLES_GENERAL".RUN_OUT_UNIT_02.CYCLE_COMPLETED AND "DB2440_GLOBAL_DATA".GLOBAL_DATA.FIX_IN_UNIT_02_STA_1_UNCLAMPED AND (("DB4000_FIX_TABLE_POSITIONS".UNIT_02.FIXTURE_1.IN_LOAD_UNLOAD_STATION_1 AND NOT "DB8000_PART_STATUS".UNIT_02.FIXTURE_1.PART_A.STATUS.PRESENT) OR ("DB4000_FIX_TABLE_POSITIONS".UNIT_02.FIXTURE_2.IN_LOAD_UNLOAD_STATION_1 AND NOT "DB8000_PART_STATUS".UNIT_02.FIXTURE_2.PART_A.STATUS.PRESENT) OR ("DB4000_FIX_TABLE_POSITIONS".UNIT_02.FIXTURE_3.IN_LOAD_UNLOAD_STATION_1 AND NOT "DB8000_PART_STATUS".UNIT_02.FIXTURE_3.PART_A.STATUS.PRESENT) OR ("DB4000_FIX_TABLE_POSITIONS".UNIT_02.FIXTURE_4.IN_LOAD_UNLOAD_STATION_1 AND NOT "DB8000_PART_STATUS".UNIT_02.FIXTURE_4.PART_A.STATUS.PRESENT)) AND "DB2440_GLOBAL_DATA".GLOBAL_DATA.UNIT_02_STA_1_AT_HOME_POS;
   "DB426_ALARMS_WARNINGS".WARNINGS."742041" := "DB1101_MACHINE_SEQUENCE".NO_PART_AT_FEED_UNIT_02;
END_REGION

REGION Network 13: MACHINE DELIVERY OCCUPIED UNIT 02
   RUNG wire#powerrail
      I_Contact( "DB8000_PART_STATUS".UNIT_02.FIXTURE_1.PART_A.STATUS.UNIT_02_STATUS.FACE_R_STATION_4_DONE )
      I_Contact( "DB8000_PART_STATUS".UNIT_02.FIXTURE_1.PART_A.STATUS.UNIT_02_STATUS.FACE_N_STATION_4_DONE )
      I_Contact( "DB8000_PART_STATUS".UNIT_02.FIXTURE_1.PART_A.STATUS.PART_REJECTED )
      Not()
      Contact( "DB4000_FIX_TABLE_POSITIONS".UNIT_02.FIXTURE_1.IN_LOAD_UNLOAD_STATION_1 )
      wire#w1
      Contact( "DB1101_MACHINE_SEQUENCE".RUNNING )
      Contact( "DB2440_GLOBAL_DATA".GLOBAL_DATA.UNIT_02_STA_1_AT_HOME_POS )
      Contact( "DB2440_GLOBAL_DATA".GLOBAL_DATA.FIX_IN_UNIT_02_STA_1_UNCLAMPED )
      wire#w2
      Coil( "DB1101_MACHINE_SEQUENCE".DELIVERY_OCCUPIED_UNIT_02 )
   END_RUNG
   RUNG wire#powerrail
      I_Contact( "DB8000_PART_STATUS".UNIT_02.FIXTURE_2.PART_A.STATUS.UNIT_02_STATUS.FACE_R_STATION_4_DONE )
      I_Contact( "DB8000_PART_STATUS".UNIT_02.FIXTURE_2.PART_A.STATUS.UNIT_02_STATUS.FACE_N_STATION_4_DONE )
      I_Contact( "DB8000_PART_STATUS".UNIT_02.FIXTURE_2.PART_A.STATUS.PART_REJECTED )
      Not()
      Contact( "DB4000_FIX_TABLE_POSITIONS".UNIT_02.FIXTURE_2.IN_LOAD_UNLOAD_STATION_1 )
   END_RUNG wire#w1
   RUNG wire#powerrail
      I_Contact( "DB8000_PART_STATUS".UNIT_02.FIXTURE_3.PART_A.STATUS.UNIT_02_STATUS.FACE_R_STATION_4_DONE )
      I_Contact( "DB8000_PART_STATUS".UNIT_02.FIXTURE_3.PART_A.STATUS.UNIT_02_STATUS.FACE_N_STATION_4_DONE )
      I_Contact( "DB8000_PART_STATUS".UNIT_02.FIXTURE_3.PART_A.STATUS.PART_REJECTED )
      Not()
      Contact( "DB4000_FIX_TABLE_POSITIONS".UNIT_02.FIXTURE_3.IN_LOAD_UNLOAD_STATION_1 )
   END_RUNG wire#w1
   RUNG wire#powerrail
      I_Contact( "DB8000_PART_STATUS".UNIT_02.FIXTURE_4.PART_A.STATUS.UNIT_02_STATUS.FACE_R_STATION_4_DONE )
      I_Contact( "DB8000_PART_STATUS".UNIT_02.FIXTURE_4.PART_A.STATUS.UNIT_02_STATUS.FACE_N_STATION_4_DONE )
      I_Contact( "DB8000_PART_STATUS".UNIT_02.FIXTURE_4.PART_A.STATUS.PART_REJECTED )
      Not()
      Contact( "DB4000_FIX_TABLE_POSITIONS".UNIT_02.FIXTURE_4.IN_LOAD_UNLOAD_STATION_1 )
   END_RUNG wire#w1
   RUNG wire#w2
      Coil( "DB426_ALARMS_WARNINGS".WARNINGS."742044" )
   END_RUNG
   // the same network as SCL:
   "DB1101_MACHINE_SEQUENCE".DELIVERY_OCCUPIED_UNIT_02 := ((NOT (NOT "DB8000_PART_STATUS".UNIT_02.FIXTURE_1.PART_A.STATUS.UNIT_02_STATUS.FACE_R_STATION_4_DONE AND NOT "DB8000_PART_STATUS".UNIT_02.FIXTURE_1.PART_A.STATUS.UNIT_02_STATUS.FACE_N_STATION_4_DONE AND NOT "DB8000_PART_STATUS".UNIT_02.FIXTURE_1.PART_A.STATUS.PART_REJECTED) AND "DB4000_FIX_TABLE_POSITIONS".UNIT_02.FIXTURE_1.IN_LOAD_UNLOAD_STATION_1) OR (NOT (NOT "DB8000_PART_STATUS".UNIT_02.FIXTURE_2.PART_A.STATUS.UNIT_02_STATUS.FACE_R_STATION_4_DONE AND NOT "DB8000_PART_STATUS".UNIT_02.FIXTURE_2.PART_A.STATUS.UNIT_02_STATUS.FACE_N_STATION_4_DONE AND NOT "DB8000_PART_STATUS".UNIT_02.FIXTURE_2.PART_A.STATUS.PART_REJECTED) AND "DB4000_FIX_TABLE_POSITIONS".UNIT_02.FIXTURE_2.IN_LOAD_UNLOAD_STATION_1) OR (NOT (NOT "DB8000_PART_STATUS".UNIT_02.FIXTURE_3.PART_A.STATUS.UNIT_02_STATUS.FACE_R_STATION_4_DONE AND NOT "DB8000_PART_STATUS".UNIT_02.FIXTURE_3.PART_A.STATUS.UNIT_02_STATUS.FACE_N_STATION_4_DONE AND NOT "DB8000_PART_STATUS".UNIT_02.FIXTURE_3.PART_A.STATUS.PART_REJECTED) AND "DB4000_FIX_TABLE_POSITIONS".UNIT_02.FIXTURE_3.IN_LOAD_UNLOAD_STATION_1) OR (NOT (NOT "DB8000_PART_STATUS".UNIT_02.FIXTURE_4.PART_A.STATUS.UNIT_02_STATUS.FACE_R_STATION_4_DONE AND NOT "DB8000_PART_STATUS".UNIT_02.FIXTURE_4.PART_A.STATUS.UNIT_02_STATUS.FACE_N_STATION_4_DONE AND NOT "DB8000_PART_STATUS".UNIT_02.FIXTURE_4.PART_A.STATUS.PART_REJECTED) AND "DB4000_FIX_TABLE_POSITIONS".UNIT_02.FIXTURE_4.IN_LOAD_UNLOAD_STATION_1)) AND "DB1101_MACHINE_SEQUENCE".RUNNING AND "DB2440_GLOBAL_DATA".GLOBAL_DATA.UNIT_02_STA_1_AT_HOME_POS AND "DB2440_GLOBAL_DATA".GLOBAL_DATA.FIX_IN_UNIT_02_STA_1_UNCLAMPED;
   "DB426_ALARMS_WARNINGS".WARNINGS."742044" := "DB1101_MACHINE_SEQUENCE".DELIVERY_OCCUPIED_UNIT_02;
END_REGION

REGION Network 14: SKIP FIXTURE UNIT 01
   // M0.3 AGREGAR SEÑALES DEL ROBOT PARA SKIP FIXTURE
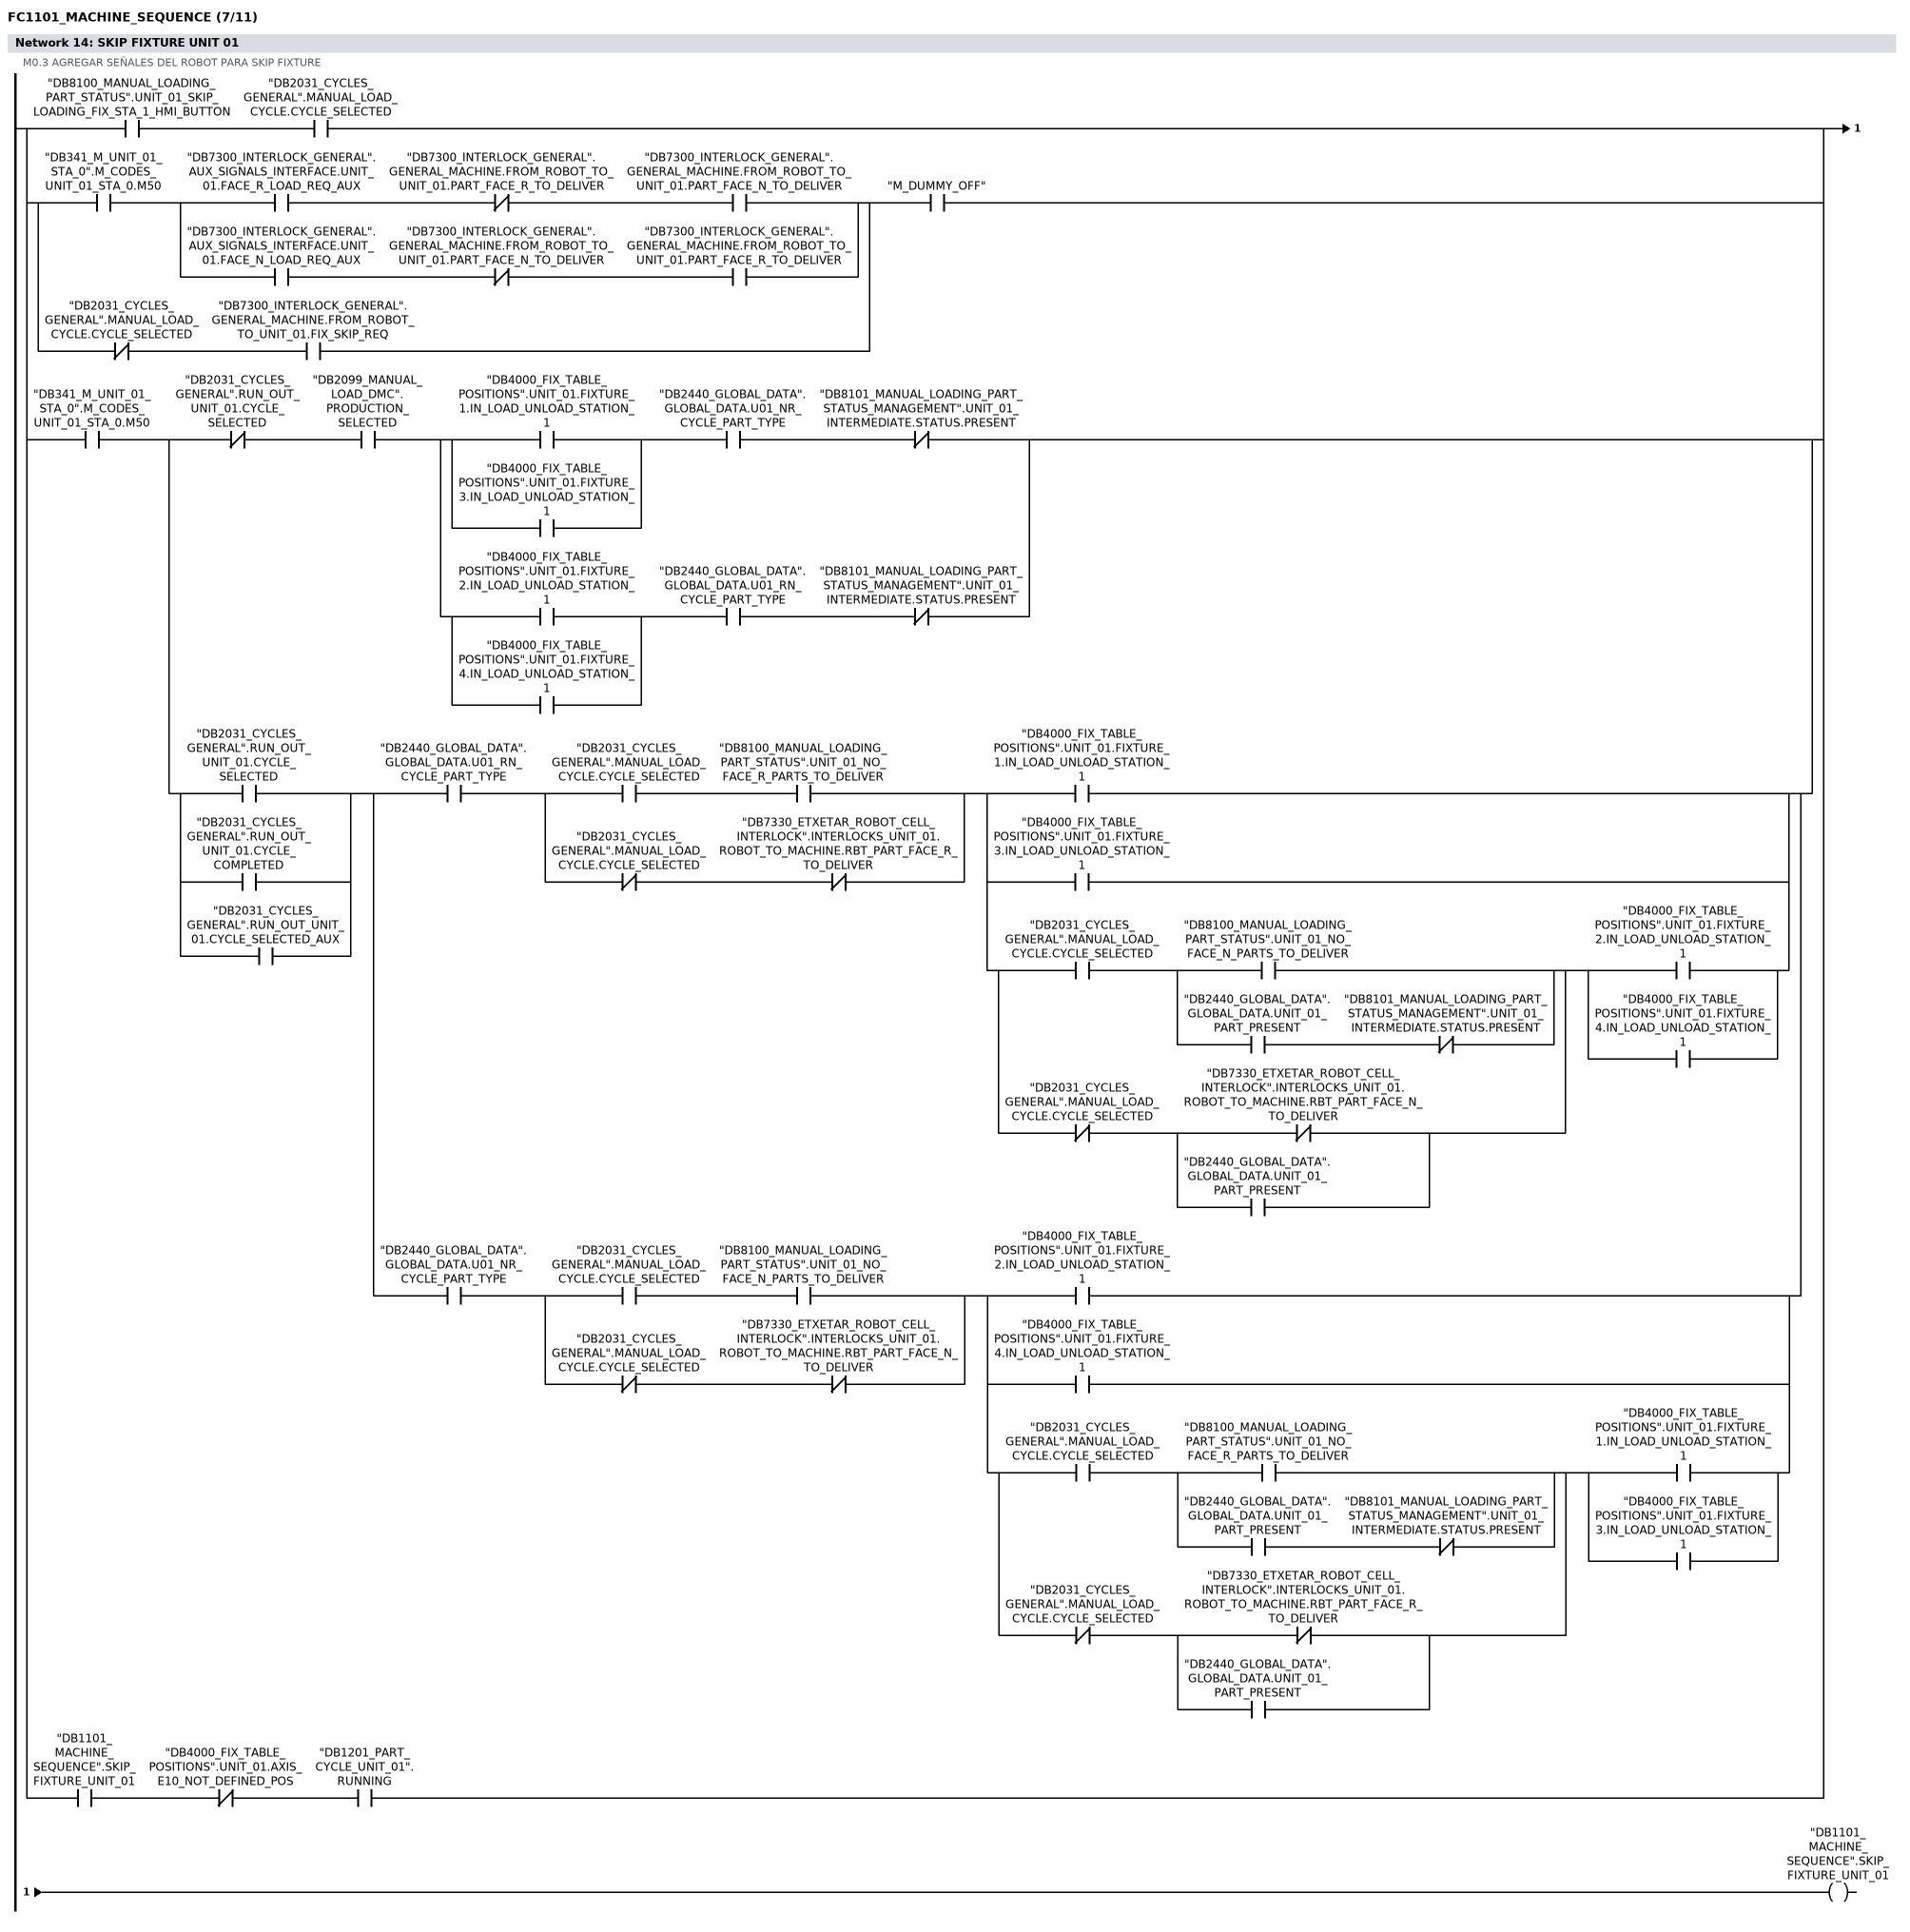
   RUNG wire#powerrail
      Contact( "DB8100_MANUAL_LOADING_PART_STATUS".UNIT_01_SKIP_LOADING_FIX_STA_1_HMI_BUTTON )
      Contact( "DB2031_CYCLES_GENERAL".MANUAL_LOAD_CYCLE.CYCLE_SELECTED )
      wire#w1
      Coil( "DB1101_MACHINE_SEQUENCE".SKIP_FIXTURE_UNIT_01 )
   END_RUNG
   RUNG wire#powerrail
      Contact( "DB341_M_UNIT_01_STA_0".M_CODES_UNIT_01_STA_0.M50 )
      wire#w2
      Contact( "DB7300_INTERLOCK_GENERAL".AUX_SIGNALS_INTERFACE.UNIT_01.FACE_R_LOAD_REQ_AUX )
      I_Contact( "DB7300_INTERLOCK_GENERAL".GENERAL_MACHINE.FROM_ROBOT_TO_UNIT_01.PART_FACE_R_TO_DELIVER )
      Contact( "DB7300_INTERLOCK_GENERAL".GENERAL_MACHINE.FROM_ROBOT_TO_UNIT_01.PART_FACE_N_TO_DELIVER )
      wire#w3
      Contact( "M_DUMMY_OFF" )
   END_RUNG wire#w1
   RUNG wire#w2
      Contact( "DB7300_INTERLOCK_GENERAL".AUX_SIGNALS_INTERFACE.UNIT_01.FACE_N_LOAD_REQ_AUX )
      I_Contact( "DB7300_INTERLOCK_GENERAL".GENERAL_MACHINE.FROM_ROBOT_TO_UNIT_01.PART_FACE_N_TO_DELIVER )
      Contact( "DB7300_INTERLOCK_GENERAL".GENERAL_MACHINE.FROM_ROBOT_TO_UNIT_01.PART_FACE_R_TO_DELIVER )
   END_RUNG wire#w3
   RUNG wire#powerrail
      I_Contact( "DB2031_CYCLES_GENERAL".MANUAL_LOAD_CYCLE.CYCLE_SELECTED )
      Contact( "DB7300_INTERLOCK_GENERAL".GENERAL_MACHINE.FROM_ROBOT_TO_UNIT_01.FIX_SKIP_REQ )
   END_RUNG wire#w3
   RUNG wire#powerrail
      Contact( "DB341_M_UNIT_01_STA_0".M_CODES_UNIT_01_STA_0.M50 )
      wire#w4
      I_Contact( "DB2031_CYCLES_GENERAL".RUN_OUT_UNIT_01.CYCLE_SELECTED )
      Contact( "DB2099_MANUAL_LOAD_DMC".PRODUCTION_SELECTED )
      wire#w5
      Contact( "DB4000_FIX_TABLE_POSITIONS".UNIT_01.FIXTURE_1.IN_LOAD_UNLOAD_STATION_1 )
      wire#w6
      Contact( "DB2440_GLOBAL_DATA".GLOBAL_DATA.U01_NR_CYCLE_PART_TYPE )
      I_Contact( "DB8101_MANUAL_LOADING_PART_STATUS_MANAGEMENT".UNIT_01_INTERMEDIATE.STATUS.PRESENT )
   END_RUNG wire#w1
   RUNG wire#w5
      Contact( "DB4000_FIX_TABLE_POSITIONS".UNIT_01.FIXTURE_3.IN_LOAD_UNLOAD_STATION_1 )
   END_RUNG wire#w6
   RUNG wire#w5
      Contact( "DB4000_FIX_TABLE_POSITIONS".UNIT_01.FIXTURE_2.IN_LOAD_UNLOAD_STATION_1 )
      wire#w7
      Contact( "DB2440_GLOBAL_DATA".GLOBAL_DATA.U01_RN_CYCLE_PART_TYPE )
      I_Contact( "DB8101_MANUAL_LOADING_PART_STATUS_MANAGEMENT".UNIT_01_INTERMEDIATE.STATUS.PRESENT )
   END_RUNG wire#w1
   RUNG wire#w5
      Contact( "DB4000_FIX_TABLE_POSITIONS".UNIT_01.FIXTURE_4.IN_LOAD_UNLOAD_STATION_1 )
   END_RUNG wire#w7
   RUNG wire#w4
      Contact( "DB2031_CYCLES_GENERAL".RUN_OUT_UNIT_01.CYCLE_SELECTED )
      wire#w8
      Contact( "DB2440_GLOBAL_DATA".GLOBAL_DATA.U01_RN_CYCLE_PART_TYPE )
      wire#w9
      Contact( "DB2031_CYCLES_GENERAL".MANUAL_LOAD_CYCLE.CYCLE_SELECTED )
      Contact( "DB8100_MANUAL_LOADING_PART_STATUS".UNIT_01_NO_FACE_R_PARTS_TO_DELIVER )
      wire#w10
      Contact( "DB4000_FIX_TABLE_POSITIONS".UNIT_01.FIXTURE_1.IN_LOAD_UNLOAD_STATION_1 )
   END_RUNG wire#w1
   RUNG wire#w4
      Contact( "DB2031_CYCLES_GENERAL".RUN_OUT_UNIT_01.CYCLE_COMPLETED )
   END_RUNG wire#w8
   RUNG wire#w4
      Contact( "DB2031_CYCLES_GENERAL".RUN_OUT_UNIT_01.CYCLE_SELECTED_AUX )
   END_RUNG wire#w8
   RUNG wire#w9
      I_Contact( "DB2031_CYCLES_GENERAL".MANUAL_LOAD_CYCLE.CYCLE_SELECTED )
      I_Contact( "DB7330_ETXETAR_ROBOT_CELL_INTERLOCK".INTERLOCKS_UNIT_01.ROBOT_TO_MACHINE.RBT_PART_FACE_R_TO_DELIVER )
   END_RUNG wire#w10
   RUNG wire#w10
      Contact( "DB4000_FIX_TABLE_POSITIONS".UNIT_01.FIXTURE_3.IN_LOAD_UNLOAD_STATION_1 )
   END_RUNG wire#w1
   RUNG wire#w10
      Contact( "DB2031_CYCLES_GENERAL".MANUAL_LOAD_CYCLE.CYCLE_SELECTED )
      wire#w11
      Contact( "DB8100_MANUAL_LOADING_PART_STATUS".UNIT_01_NO_FACE_N_PARTS_TO_DELIVER )
      wire#w12
      Contact( "DB4000_FIX_TABLE_POSITIONS".UNIT_01.FIXTURE_2.IN_LOAD_UNLOAD_STATION_1 )
   END_RUNG wire#w1
   RUNG wire#w11
      Contact( "DB2440_GLOBAL_DATA".GLOBAL_DATA.UNIT_01_PART_PRESENT )
      I_Contact( "DB8101_MANUAL_LOADING_PART_STATUS_MANAGEMENT".UNIT_01_INTERMEDIATE.STATUS.PRESENT )
   END_RUNG wire#w12
   RUNG wire#w10
      I_Contact( "DB2031_CYCLES_GENERAL".MANUAL_LOAD_CYCLE.CYCLE_SELECTED )
      wire#w13
      I_Contact( "DB7330_ETXETAR_ROBOT_CELL_INTERLOCK".INTERLOCKS_UNIT_01.ROBOT_TO_MACHINE.RBT_PART_FACE_N_TO_DELIVER )
   END_RUNG wire#w12
   RUNG wire#w13
      Contact( "DB2440_GLOBAL_DATA".GLOBAL_DATA.UNIT_01_PART_PRESENT )
   END_RUNG wire#w12
   RUNG wire#w12
      Contact( "DB4000_FIX_TABLE_POSITIONS".UNIT_01.FIXTURE_4.IN_LOAD_UNLOAD_STATION_1 )
   END_RUNG wire#w1
   RUNG wire#w8
      Contact( "DB2440_GLOBAL_DATA".GLOBAL_DATA.U01_NR_CYCLE_PART_TYPE )
      wire#w14
      Contact( "DB2031_CYCLES_GENERAL".MANUAL_LOAD_CYCLE.CYCLE_SELECTED )
      Contact( "DB8100_MANUAL_LOADING_PART_STATUS".UNIT_01_NO_FACE_N_PARTS_TO_DELIVER )
      wire#w15
      Contact( "DB4000_FIX_TABLE_POSITIONS".UNIT_01.FIXTURE_2.IN_LOAD_UNLOAD_STATION_1 )
   END_RUNG wire#w1
   RUNG wire#w14
      I_Contact( "DB2031_CYCLES_GENERAL".MANUAL_LOAD_CYCLE.CYCLE_SELECTED )
      I_Contact( "DB7330_ETXETAR_ROBOT_CELL_INTERLOCK".INTERLOCKS_UNIT_01.ROBOT_TO_MACHINE.RBT_PART_FACE_N_TO_DELIVER )
   END_RUNG wire#w15
   RUNG wire#w15
      Contact( "DB4000_FIX_TABLE_POSITIONS".UNIT_01.FIXTURE_4.IN_LOAD_UNLOAD_STATION_1 )
   END_RUNG wire#w1
   RUNG wire#w15
      Contact( "DB2031_CYCLES_GENERAL".MANUAL_LOAD_CYCLE.CYCLE_SELECTED )
      wire#w16
      Contact( "DB8100_MANUAL_LOADING_PART_STATUS".UNIT_01_NO_FACE_R_PARTS_TO_DELIVER )
      wire#w17
      Contact( "DB4000_FIX_TABLE_POSITIONS".UNIT_01.FIXTURE_1.IN_LOAD_UNLOAD_STATION_1 )
   END_RUNG wire#w1
   RUNG wire#w16
      Contact( "DB2440_GLOBAL_DATA".GLOBAL_DATA.UNIT_01_PART_PRESENT )
      I_Contact( "DB8101_MANUAL_LOADING_PART_STATUS_MANAGEMENT".UNIT_01_INTERMEDIATE.STATUS.PRESENT )
   END_RUNG wire#w17
   RUNG wire#w15
      I_Contact( "DB2031_CYCLES_GENERAL".MANUAL_LOAD_CYCLE.CYCLE_SELECTED )
      wire#w18
      I_Contact( "DB7330_ETXETAR_ROBOT_CELL_INTERLOCK".INTERLOCKS_UNIT_01.ROBOT_TO_MACHINE.RBT_PART_FACE_R_TO_DELIVER )
   END_RUNG wire#w17
   RUNG wire#w18
      Contact( "DB2440_GLOBAL_DATA".GLOBAL_DATA.UNIT_01_PART_PRESENT )
   END_RUNG wire#w17
   RUNG wire#w17
      Contact( "DB4000_FIX_TABLE_POSITIONS".UNIT_01.FIXTURE_3.IN_LOAD_UNLOAD_STATION_1 )
   END_RUNG wire#w1
   RUNG wire#powerrail
      Contact( "DB1101_MACHINE_SEQUENCE".SKIP_FIXTURE_UNIT_01 )
      I_Contact( "DB4000_FIX_TABLE_POSITIONS".UNIT_01.AXIS_E10_NOT_DEFINED_POS )
      Contact( "DB1201_PART_CYCLE_UNIT_01".RUNNING )
   END_RUNG wire#w1
   // the same network as SCL:
   "DB1101_MACHINE_SEQUENCE".SKIP_FIXTURE_UNIT_01 := ("DB8100_MANUAL_LOADING_PART_STATUS".UNIT_01_SKIP_LOADING_FIX_STA_1_HMI_BUTTON AND "DB2031_CYCLES_GENERAL".MANUAL_LOAD_CYCLE.CYCLE_SELECTED) OR ((("DB341_M_UNIT_01_STA_0".M_CODES_UNIT_01_STA_0.M50 AND (("DB7300_INTERLOCK_GENERAL".AUX_SIGNALS_INTERFACE.UNIT_01.FACE_R_LOAD_REQ_AUX AND NOT "DB7300_INTERLOCK_GENERAL".GENERAL_MACHINE.FROM_ROBOT_TO_UNIT_01.PART_FACE_R_TO_DELIVER AND "DB7300_INTERLOCK_GENERAL".GENERAL_MACHINE.FROM_ROBOT_TO_UNIT_01.PART_FACE_N_TO_DELIVER) OR ("DB7300_INTERLOCK_GENERAL".AUX_SIGNALS_INTERFACE.UNIT_01.FACE_N_LOAD_REQ_AUX AND NOT "DB7300_INTERLOCK_GENERAL".GENERAL_MACHINE.FROM_ROBOT_TO_UNIT_01.PART_FACE_N_TO_DELIVER AND "DB7300_INTERLOCK_GENERAL".GENERAL_MACHINE.FROM_ROBOT_TO_UNIT_01.PART_FACE_R_TO_DELIVER))) OR (NOT "DB2031_CYCLES_GENERAL".MANUAL_LOAD_CYCLE.CYCLE_SELECTED AND "DB7300_INTERLOCK_GENERAL".GENERAL_MACHINE.FROM_ROBOT_TO_UNIT_01.FIX_SKIP_REQ)) AND "M_DUMMY_OFF") OR ("DB341_M_UNIT_01_STA_0".M_CODES_UNIT_01_STA_0.M50 AND ((NOT "DB2031_CYCLES_GENERAL".RUN_OUT_UNIT_01.CYCLE_SELECTED AND "DB2099_MANUAL_LOAD_DMC".PRODUCTION_SELECTED AND ((("DB4000_FIX_TABLE_POSITIONS".UNIT_01.FIXTURE_1.IN_LOAD_UNLOAD_STATION_1 OR "DB4000_FIX_TABLE_POSITIONS".UNIT_01.FIXTURE_3.IN_LOAD_UNLOAD_STATION_1) AND "DB2440_GLOBAL_DATA".GLOBAL_DATA.U01_NR_CYCLE_PART_TYPE AND NOT "DB8101_MANUAL_LOADING_PART_STATUS_MANAGEMENT".UNIT_01_INTERMEDIATE.STATUS.PRESENT) OR (("DB4000_FIX_TABLE_POSITIONS".UNIT_01.FIXTURE_2.IN_LOAD_UNLOAD_STATION_1 OR "DB4000_FIX_TABLE_POSITIONS".UNIT_01.FIXTURE_4.IN_LOAD_UNLOAD_STATION_1) AND "DB2440_GLOBAL_DATA".GLOBAL_DATA.U01_RN_CYCLE_PART_TYPE AND NOT "DB8101_MANUAL_LOADING_PART_STATUS_MANAGEMENT".UNIT_01_INTERMEDIATE.STATUS.PRESENT))) OR (("DB2031_CYCLES_GENERAL".RUN_OUT_UNIT_01.CYCLE_SELECTED OR "DB2031_CYCLES_GENERAL".RUN_OUT_UNIT_01.CYCLE_COMPLETED OR "DB2031_CYCLES_GENERAL".RUN_OUT_UNIT_01.CYCLE_SELECTED_AUX) AND (("DB2440_GLOBAL_DATA".GLOBAL_DATA.U01_RN_CYCLE_PART_TYPE AND (("DB2031_CYCLES_GENERAL".MANUAL_LOAD_CYCLE.CYCLE_SELECTED AND "DB8100_MANUAL_LOADING_PART_STATUS".UNIT_01_NO_FACE_R_PARTS_TO_DELIVER) OR (NOT "DB2031_CYCLES_GENERAL".MANUAL_LOAD_CYCLE.CYCLE_SELECTED AND NOT "DB7330_ETXETAR_ROBOT_CELL_INTERLOCK".INTERLOCKS_UNIT_01.ROBOT_TO_MACHINE.RBT_PART_FACE_R_TO_DELIVER)) AND ("DB4000_FIX_TABLE_POSITIONS".UNIT_01.FIXTURE_1.IN_LOAD_UNLOAD_STATION_1 OR "DB4000_FIX_TABLE_POSITIONS".UNIT_01.FIXTURE_3.IN_LOAD_UNLOAD_STATION_1 OR ((("DB2031_CYCLES_GENERAL".MANUAL_LOAD_CYCLE.CYCLE_SELECTED AND ("DB8100_MANUAL_LOADING_PART_STATUS".UNIT_01_NO_FACE_N_PARTS_TO_DELIVER OR ("DB2440_GLOBAL_DATA".GLOBAL_DATA.UNIT_01_PART_PRESENT AND NOT "DB8101_MANUAL_LOADING_PART_STATUS_MANAGEMENT".UNIT_01_INTERMEDIATE.STATUS.PRESENT))) OR (NOT "DB2031_CYCLES_GENERAL".MANUAL_LOAD_CYCLE.CYCLE_SELECTED AND (NOT "DB7330_ETXETAR_ROBOT_CELL_INTERLOCK".INTERLOCKS_UNIT_01.ROBOT_TO_MACHINE.RBT_PART_FACE_N_TO_DELIVER OR "DB2440_GLOBAL_DATA".GLOBAL_DATA.UNIT_01_PART_PRESENT))) AND ("DB4000_FIX_TABLE_POSITIONS".UNIT_01.FIXTURE_2.IN_LOAD_UNLOAD_STATION_1 OR "DB4000_FIX_TABLE_POSITIONS".UNIT_01.FIXTURE_4.IN_LOAD_UNLOAD_STATION_1)))) OR ("DB2440_GLOBAL_DATA".GLOBAL_DATA.U01_NR_CYCLE_PART_TYPE AND (("DB2031_CYCLES_GENERAL".MANUAL_LOAD_CYCLE.CYCLE_SELECTED AND "DB8100_MANUAL_LOADING_PART_STATUS".UNIT_01_NO_FACE_N_PARTS_TO_DELIVER) OR (NOT "DB2031_CYCLES_GENERAL".MANUAL_LOAD_CYCLE.CYCLE_SELECTED AND NOT "DB7330_ETXETAR_ROBOT_CELL_INTERLOCK".INTERLOCKS_UNIT_01.ROBOT_TO_MACHINE.RBT_PART_FACE_N_TO_DELIVER)) AND ("DB4000_FIX_TABLE_POSITIONS".UNIT_01.FIXTURE_2.IN_LOAD_UNLOAD_STATION_1 OR "DB4000_FIX_TABLE_POSITIONS".UNIT_01.FIXTURE_4.IN_LOAD_UNLOAD_STATION_1 OR ((("DB2031_CYCLES_GENERAL".MANUAL_LOAD_CYCLE.CYCLE_SELECTED AND ("DB8100_MANUAL_LOADING_PART_STATUS".UNIT_01_NO_FACE_R_PARTS_TO_DELIVER OR ("DB2440_GLOBAL_DATA".GLOBAL_DATA.UNIT_01_PART_PRESENT AND NOT "DB8101_MANUAL_LOADING_PART_STATUS_MANAGEMENT".UNIT_01_INTERMEDIATE.STATUS.PRESENT))) OR (NOT "DB2031_CYCLES_GENERAL".MANUAL_LOAD_CYCLE.CYCLE_SELECTED AND (NOT "DB7330_ETXETAR_ROBOT_CELL_INTERLOCK".INTERLOCKS_UNIT_01.ROBOT_TO_MACHINE.RBT_PART_FACE_R_TO_DELIVER OR "DB2440_GLOBAL_DATA".GLOBAL_DATA.UNIT_01_PART_PRESENT))) AND ("DB4000_FIX_TABLE_POSITIONS".UNIT_01.FIXTURE_1.IN_LOAD_UNLOAD_STATION_1 OR "DB4000_FIX_TABLE_POSITIONS".UNIT_01.FIXTURE_3.IN_LOAD_UNLOAD_STATION_1)))))))) OR ("DB1101_MACHINE_SEQUENCE".SKIP_FIXTURE_UNIT_01 AND NOT "DB4000_FIX_TABLE_POSITIONS".UNIT_01.AXIS_E10_NOT_DEFINED_POS AND "DB1201_PART_CYCLE_UNIT_01".RUNNING);
END_REGION

REGION Network 15: SKIP FIXTURE UNIT 02
   // M0.3 AGREGAR SEÑALES DEL ROBOT PARA SKIP FIXTURE
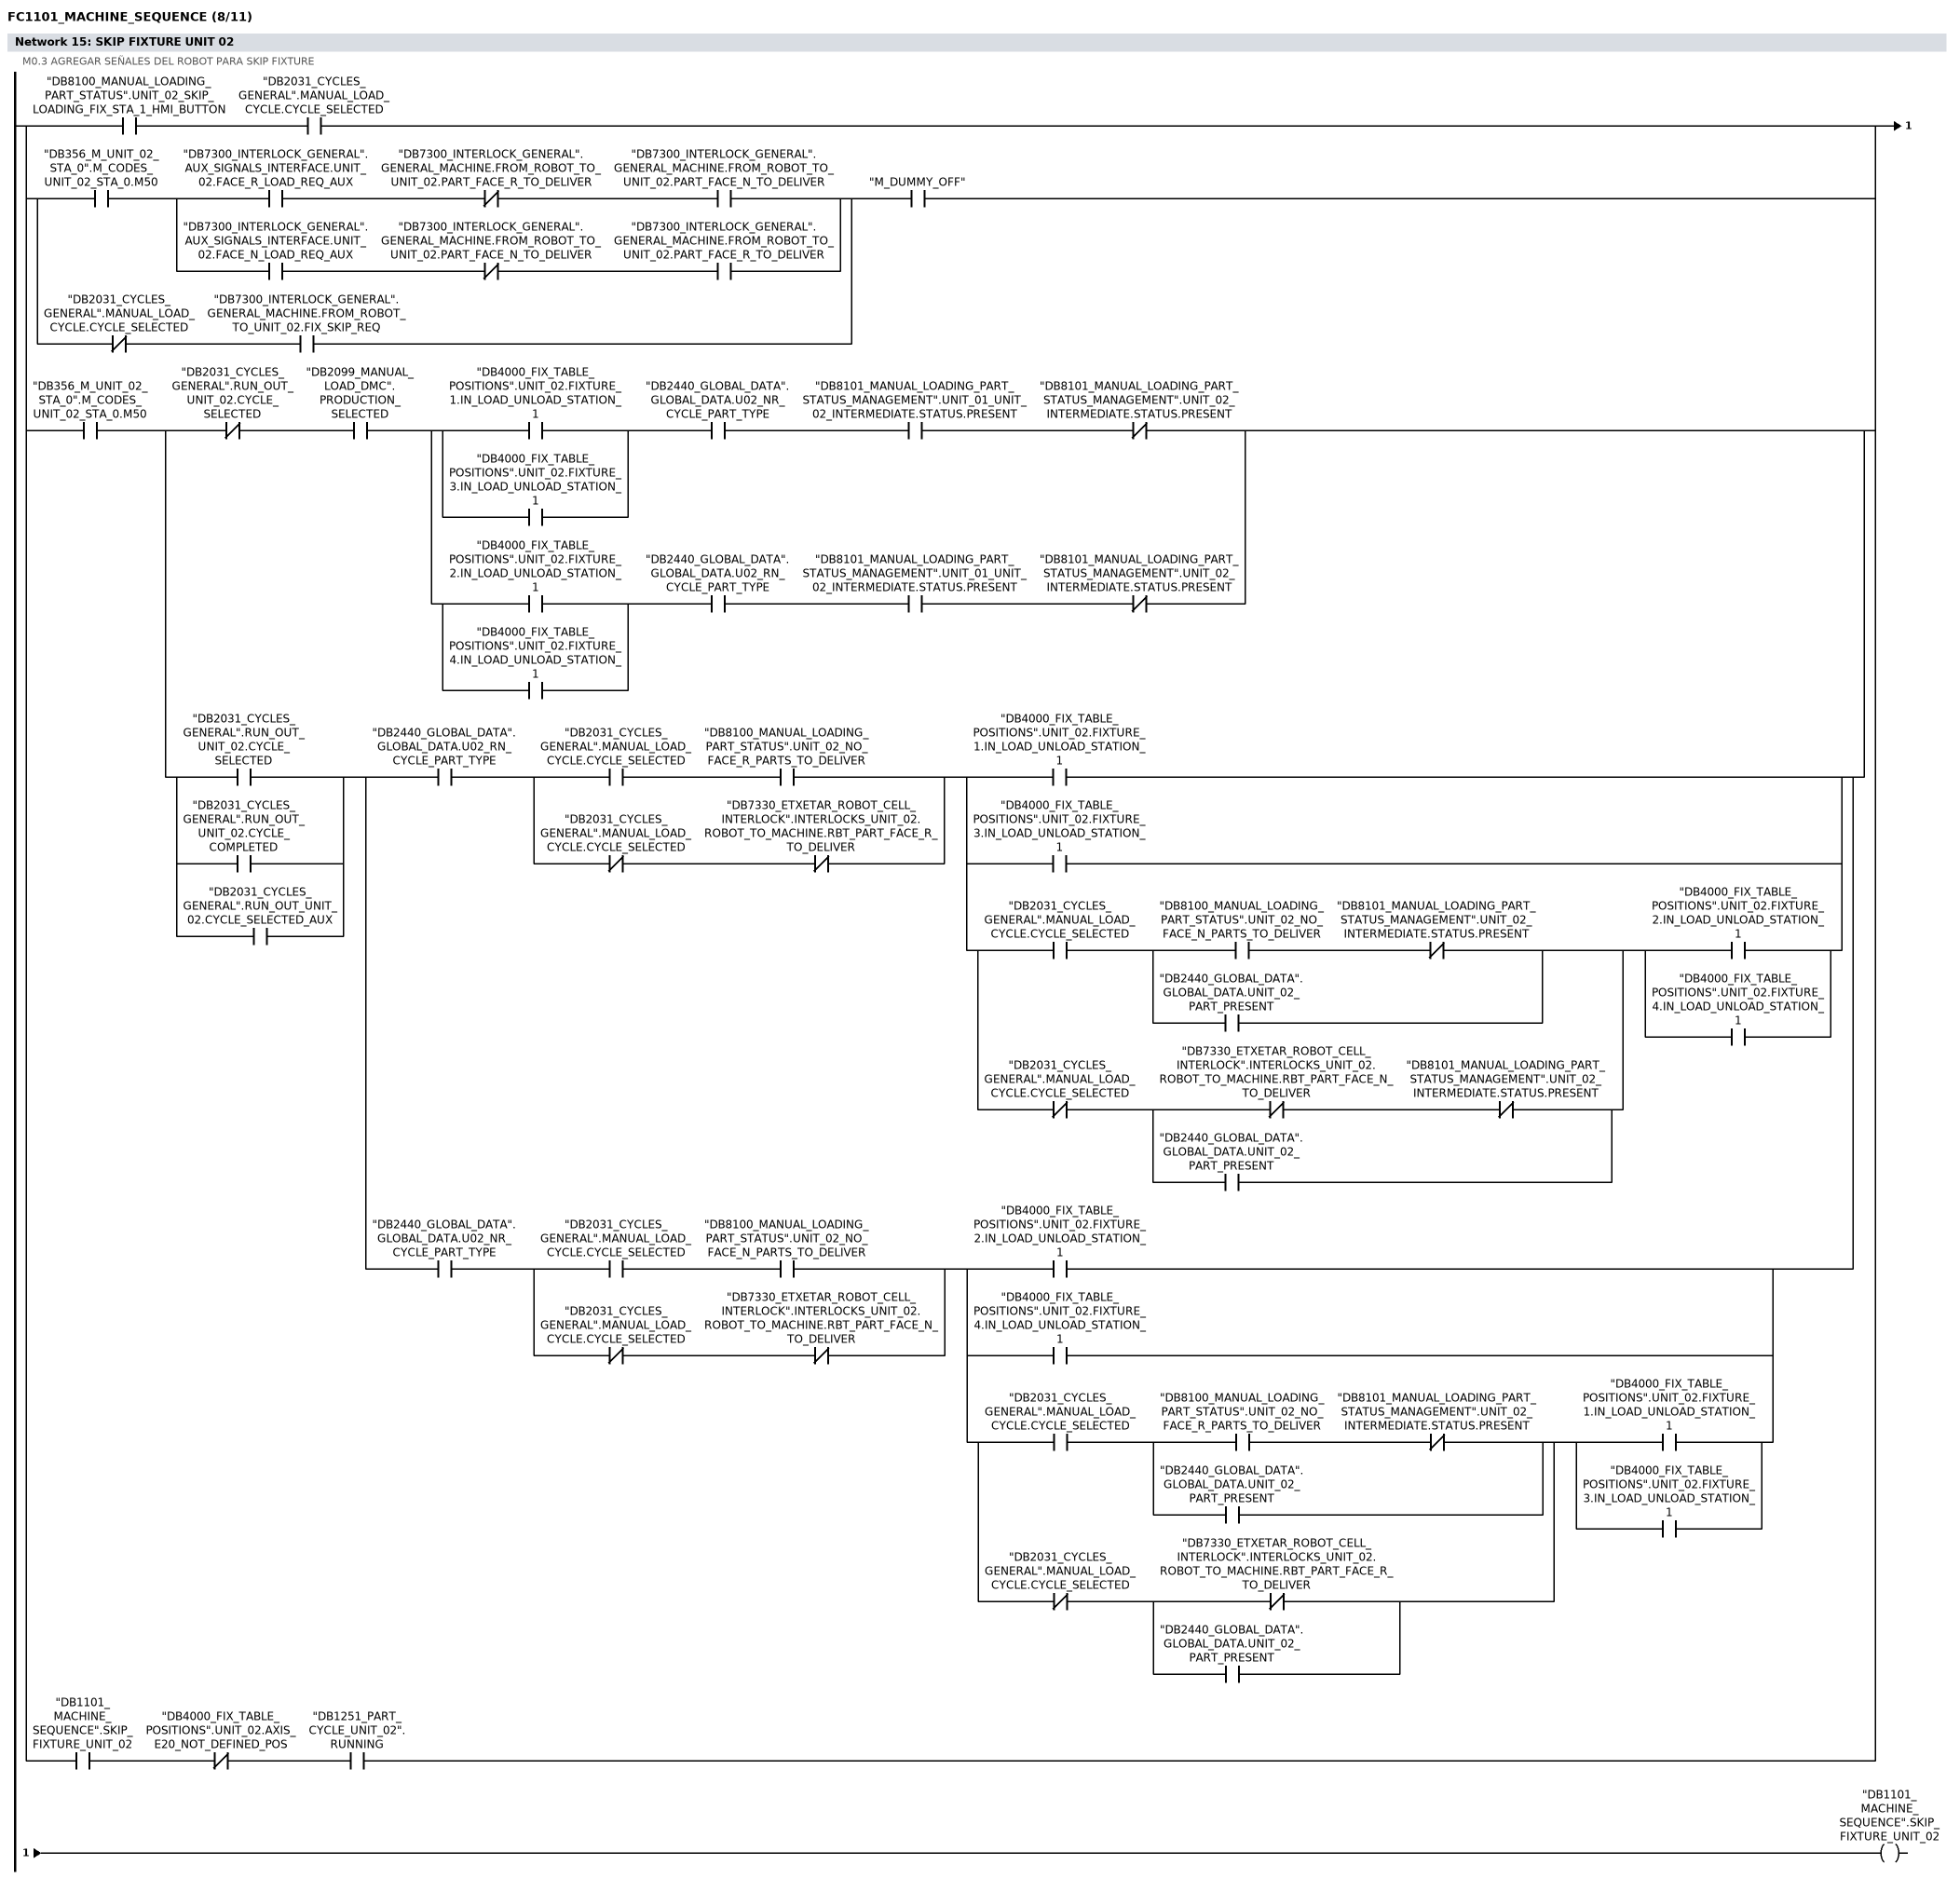
   RUNG wire#powerrail
      Contact( "DB8100_MANUAL_LOADING_PART_STATUS".UNIT_02_SKIP_LOADING_FIX_STA_1_HMI_BUTTON )
      Contact( "DB2031_CYCLES_GENERAL".MANUAL_LOAD_CYCLE.CYCLE_SELECTED )
      wire#w1
      Coil( "DB1101_MACHINE_SEQUENCE".SKIP_FIXTURE_UNIT_02 )
   END_RUNG
   RUNG wire#powerrail
      Contact( "DB356_M_UNIT_02_STA_0".M_CODES_UNIT_02_STA_0.M50 )
      wire#w2
      Contact( "DB7300_INTERLOCK_GENERAL".AUX_SIGNALS_INTERFACE.UNIT_02.FACE_R_LOAD_REQ_AUX )
      I_Contact( "DB7300_INTERLOCK_GENERAL".GENERAL_MACHINE.FROM_ROBOT_TO_UNIT_02.PART_FACE_R_TO_DELIVER )
      Contact( "DB7300_INTERLOCK_GENERAL".GENERAL_MACHINE.FROM_ROBOT_TO_UNIT_02.PART_FACE_N_TO_DELIVER )
      wire#w3
      Contact( "M_DUMMY_OFF" )
   END_RUNG wire#w1
   RUNG wire#w2
      Contact( "DB7300_INTERLOCK_GENERAL".AUX_SIGNALS_INTERFACE.UNIT_02.FACE_N_LOAD_REQ_AUX )
      I_Contact( "DB7300_INTERLOCK_GENERAL".GENERAL_MACHINE.FROM_ROBOT_TO_UNIT_02.PART_FACE_N_TO_DELIVER )
      Contact( "DB7300_INTERLOCK_GENERAL".GENERAL_MACHINE.FROM_ROBOT_TO_UNIT_02.PART_FACE_R_TO_DELIVER )
   END_RUNG wire#w3
   RUNG wire#powerrail
      I_Contact( "DB2031_CYCLES_GENERAL".MANUAL_LOAD_CYCLE.CYCLE_SELECTED )
      Contact( "DB7300_INTERLOCK_GENERAL".GENERAL_MACHINE.FROM_ROBOT_TO_UNIT_02.FIX_SKIP_REQ )
   END_RUNG wire#w3
   RUNG wire#powerrail
      Contact( "DB356_M_UNIT_02_STA_0".M_CODES_UNIT_02_STA_0.M50 )
      wire#w4
      I_Contact( "DB2031_CYCLES_GENERAL".RUN_OUT_UNIT_02.CYCLE_SELECTED )
      Contact( "DB2099_MANUAL_LOAD_DMC".PRODUCTION_SELECTED )
      wire#w5
      Contact( "DB4000_FIX_TABLE_POSITIONS".UNIT_02.FIXTURE_1.IN_LOAD_UNLOAD_STATION_1 )
      wire#w6
      Contact( "DB2440_GLOBAL_DATA".GLOBAL_DATA.U02_NR_CYCLE_PART_TYPE )
      Contact( "DB8101_MANUAL_LOADING_PART_STATUS_MANAGEMENT".UNIT_01_UNIT_02_INTERMEDIATE.STATUS.PRESENT )
      I_Contact( "DB8101_MANUAL_LOADING_PART_STATUS_MANAGEMENT".UNIT_02_INTERMEDIATE.STATUS.PRESENT )
   END_RUNG wire#w1
   RUNG wire#w5
      Contact( "DB4000_FIX_TABLE_POSITIONS".UNIT_02.FIXTURE_3.IN_LOAD_UNLOAD_STATION_1 )
   END_RUNG wire#w6
   RUNG wire#w5
      Contact( "DB4000_FIX_TABLE_POSITIONS".UNIT_02.FIXTURE_2.IN_LOAD_UNLOAD_STATION_1 )
      wire#w7
      Contact( "DB2440_GLOBAL_DATA".GLOBAL_DATA.U02_RN_CYCLE_PART_TYPE )
      Contact( "DB8101_MANUAL_LOADING_PART_STATUS_MANAGEMENT".UNIT_01_UNIT_02_INTERMEDIATE.STATUS.PRESENT )
      I_Contact( "DB8101_MANUAL_LOADING_PART_STATUS_MANAGEMENT".UNIT_02_INTERMEDIATE.STATUS.PRESENT )
   END_RUNG wire#w1
   RUNG wire#w5
      Contact( "DB4000_FIX_TABLE_POSITIONS".UNIT_02.FIXTURE_4.IN_LOAD_UNLOAD_STATION_1 )
   END_RUNG wire#w7
   RUNG wire#w4
      Contact( "DB2031_CYCLES_GENERAL".RUN_OUT_UNIT_02.CYCLE_SELECTED )
      wire#w8
      Contact( "DB2440_GLOBAL_DATA".GLOBAL_DATA.U02_RN_CYCLE_PART_TYPE )
      wire#w9
      Contact( "DB2031_CYCLES_GENERAL".MANUAL_LOAD_CYCLE.CYCLE_SELECTED )
      Contact( "DB8100_MANUAL_LOADING_PART_STATUS".UNIT_02_NO_FACE_R_PARTS_TO_DELIVER )
      wire#w10
      Contact( "DB4000_FIX_TABLE_POSITIONS".UNIT_02.FIXTURE_1.IN_LOAD_UNLOAD_STATION_1 )
   END_RUNG wire#w1
   RUNG wire#w4
      Contact( "DB2031_CYCLES_GENERAL".RUN_OUT_UNIT_02.CYCLE_COMPLETED )
   END_RUNG wire#w8
   RUNG wire#w4
      Contact( "DB2031_CYCLES_GENERAL".RUN_OUT_UNIT_02.CYCLE_SELECTED_AUX )
   END_RUNG wire#w8
   RUNG wire#w9
      I_Contact( "DB2031_CYCLES_GENERAL".MANUAL_LOAD_CYCLE.CYCLE_SELECTED )
      I_Contact( "DB7330_ETXETAR_ROBOT_CELL_INTERLOCK".INTERLOCKS_UNIT_02.ROBOT_TO_MACHINE.RBT_PART_FACE_R_TO_DELIVER )
   END_RUNG wire#w10
   RUNG wire#w10
      Contact( "DB4000_FIX_TABLE_POSITIONS".UNIT_02.FIXTURE_3.IN_LOAD_UNLOAD_STATION_1 )
   END_RUNG wire#w1
   RUNG wire#w10
      Contact( "DB2031_CYCLES_GENERAL".MANUAL_LOAD_CYCLE.CYCLE_SELECTED )
      wire#w11
      Contact( "DB8100_MANUAL_LOADING_PART_STATUS".UNIT_02_NO_FACE_N_PARTS_TO_DELIVER )
      I_Contact( "DB8101_MANUAL_LOADING_PART_STATUS_MANAGEMENT".UNIT_02_INTERMEDIATE.STATUS.PRESENT )
      wire#w12
      Contact( "DB4000_FIX_TABLE_POSITIONS".UNIT_02.FIXTURE_2.IN_LOAD_UNLOAD_STATION_1 )
   END_RUNG wire#w1
   RUNG wire#w11
      Contact( "DB2440_GLOBAL_DATA".GLOBAL_DATA.UNIT_02_PART_PRESENT )
   END_RUNG wire#w12
   RUNG wire#w10
      I_Contact( "DB2031_CYCLES_GENERAL".MANUAL_LOAD_CYCLE.CYCLE_SELECTED )
      wire#w13
      I_Contact( "DB7330_ETXETAR_ROBOT_CELL_INTERLOCK".INTERLOCKS_UNIT_02.ROBOT_TO_MACHINE.RBT_PART_FACE_N_TO_DELIVER )
      I_Contact( "DB8101_MANUAL_LOADING_PART_STATUS_MANAGEMENT".UNIT_02_INTERMEDIATE.STATUS.PRESENT )
   END_RUNG wire#w12
   RUNG wire#w13
      Contact( "DB2440_GLOBAL_DATA".GLOBAL_DATA.UNIT_02_PART_PRESENT )
   END_RUNG wire#w12
   RUNG wire#w12
      Contact( "DB4000_FIX_TABLE_POSITIONS".UNIT_02.FIXTURE_4.IN_LOAD_UNLOAD_STATION_1 )
   END_RUNG wire#w1
   RUNG wire#w8
      Contact( "DB2440_GLOBAL_DATA".GLOBAL_DATA.U02_NR_CYCLE_PART_TYPE )
      wire#w14
      Contact( "DB2031_CYCLES_GENERAL".MANUAL_LOAD_CYCLE.CYCLE_SELECTED )
      Contact( "DB8100_MANUAL_LOADING_PART_STATUS".UNIT_02_NO_FACE_N_PARTS_TO_DELIVER )
      wire#w15
      Contact( "DB4000_FIX_TABLE_POSITIONS".UNIT_02.FIXTURE_2.IN_LOAD_UNLOAD_STATION_1 )
   END_RUNG wire#w1
   RUNG wire#w14
      I_Contact( "DB2031_CYCLES_GENERAL".MANUAL_LOAD_CYCLE.CYCLE_SELECTED )
      I_Contact( "DB7330_ETXETAR_ROBOT_CELL_INTERLOCK".INTERLOCKS_UNIT_02.ROBOT_TO_MACHINE.RBT_PART_FACE_N_TO_DELIVER )
   END_RUNG wire#w15
   RUNG wire#w15
      Contact( "DB4000_FIX_TABLE_POSITIONS".UNIT_02.FIXTURE_4.IN_LOAD_UNLOAD_STATION_1 )
   END_RUNG wire#w1
   RUNG wire#w15
      Contact( "DB2031_CYCLES_GENERAL".MANUAL_LOAD_CYCLE.CYCLE_SELECTED )
      wire#w16
      Contact( "DB8100_MANUAL_LOADING_PART_STATUS".UNIT_02_NO_FACE_R_PARTS_TO_DELIVER )
      I_Contact( "DB8101_MANUAL_LOADING_PART_STATUS_MANAGEMENT".UNIT_02_INTERMEDIATE.STATUS.PRESENT )
      wire#w17
      Contact( "DB4000_FIX_TABLE_POSITIONS".UNIT_02.FIXTURE_1.IN_LOAD_UNLOAD_STATION_1 )
   END_RUNG wire#w1
   RUNG wire#w16
      Contact( "DB2440_GLOBAL_DATA".GLOBAL_DATA.UNIT_02_PART_PRESENT )
   END_RUNG wire#w17
   RUNG wire#w15
      I_Contact( "DB2031_CYCLES_GENERAL".MANUAL_LOAD_CYCLE.CYCLE_SELECTED )
      wire#w18
      I_Contact( "DB7330_ETXETAR_ROBOT_CELL_INTERLOCK".INTERLOCKS_UNIT_02.ROBOT_TO_MACHINE.RBT_PART_FACE_R_TO_DELIVER )
   END_RUNG wire#w17
   RUNG wire#w18
      Contact( "DB2440_GLOBAL_DATA".GLOBAL_DATA.UNIT_02_PART_PRESENT )
   END_RUNG wire#w17
   RUNG wire#w17
      Contact( "DB4000_FIX_TABLE_POSITIONS".UNIT_02.FIXTURE_3.IN_LOAD_UNLOAD_STATION_1 )
   END_RUNG wire#w1
   RUNG wire#powerrail
      Contact( "DB1101_MACHINE_SEQUENCE".SKIP_FIXTURE_UNIT_02 )
      I_Contact( "DB4000_FIX_TABLE_POSITIONS".UNIT_02.AXIS_E20_NOT_DEFINED_POS )
      Contact( "DB1251_PART_CYCLE_UNIT_02".RUNNING )
   END_RUNG wire#w1
   // the same network as SCL:
   "DB1101_MACHINE_SEQUENCE".SKIP_FIXTURE_UNIT_02 := ("DB8100_MANUAL_LOADING_PART_STATUS".UNIT_02_SKIP_LOADING_FIX_STA_1_HMI_BUTTON AND "DB2031_CYCLES_GENERAL".MANUAL_LOAD_CYCLE.CYCLE_SELECTED) OR ((("DB356_M_UNIT_02_STA_0".M_CODES_UNIT_02_STA_0.M50 AND (("DB7300_INTERLOCK_GENERAL".AUX_SIGNALS_INTERFACE.UNIT_02.FACE_R_LOAD_REQ_AUX AND NOT "DB7300_INTERLOCK_GENERAL".GENERAL_MACHINE.FROM_ROBOT_TO_UNIT_02.PART_FACE_R_TO_DELIVER AND "DB7300_INTERLOCK_GENERAL".GENERAL_MACHINE.FROM_ROBOT_TO_UNIT_02.PART_FACE_N_TO_DELIVER) OR ("DB7300_INTERLOCK_GENERAL".AUX_SIGNALS_INTERFACE.UNIT_02.FACE_N_LOAD_REQ_AUX AND NOT "DB7300_INTERLOCK_GENERAL".GENERAL_MACHINE.FROM_ROBOT_TO_UNIT_02.PART_FACE_N_TO_DELIVER AND "DB7300_INTERLOCK_GENERAL".GENERAL_MACHINE.FROM_ROBOT_TO_UNIT_02.PART_FACE_R_TO_DELIVER))) OR (NOT "DB2031_CYCLES_GENERAL".MANUAL_LOAD_CYCLE.CYCLE_SELECTED AND "DB7300_INTERLOCK_GENERAL".GENERAL_MACHINE.FROM_ROBOT_TO_UNIT_02.FIX_SKIP_REQ)) AND "M_DUMMY_OFF") OR ("DB356_M_UNIT_02_STA_0".M_CODES_UNIT_02_STA_0.M50 AND ((NOT "DB2031_CYCLES_GENERAL".RUN_OUT_UNIT_02.CYCLE_SELECTED AND "DB2099_MANUAL_LOAD_DMC".PRODUCTION_SELECTED AND ((("DB4000_FIX_TABLE_POSITIONS".UNIT_02.FIXTURE_1.IN_LOAD_UNLOAD_STATION_1 OR "DB4000_FIX_TABLE_POSITIONS".UNIT_02.FIXTURE_3.IN_LOAD_UNLOAD_STATION_1) AND "DB2440_GLOBAL_DATA".GLOBAL_DATA.U02_NR_CYCLE_PART_TYPE AND "DB8101_MANUAL_LOADING_PART_STATUS_MANAGEMENT".UNIT_01_UNIT_02_INTERMEDIATE.STATUS.PRESENT AND NOT "DB8101_MANUAL_LOADING_PART_STATUS_MANAGEMENT".UNIT_02_INTERMEDIATE.STATUS.PRESENT) OR (("DB4000_FIX_TABLE_POSITIONS".UNIT_02.FIXTURE_2.IN_LOAD_UNLOAD_STATION_1 OR "DB4000_FIX_TABLE_POSITIONS".UNIT_02.FIXTURE_4.IN_LOAD_UNLOAD_STATION_1) AND "DB2440_GLOBAL_DATA".GLOBAL_DATA.U02_RN_CYCLE_PART_TYPE AND "DB8101_MANUAL_LOADING_PART_STATUS_MANAGEMENT".UNIT_01_UNIT_02_INTERMEDIATE.STATUS.PRESENT AND NOT "DB8101_MANUAL_LOADING_PART_STATUS_MANAGEMENT".UNIT_02_INTERMEDIATE.STATUS.PRESENT))) OR (("DB2031_CYCLES_GENERAL".RUN_OUT_UNIT_02.CYCLE_SELECTED OR "DB2031_CYCLES_GENERAL".RUN_OUT_UNIT_02.CYCLE_COMPLETED OR "DB2031_CYCLES_GENERAL".RUN_OUT_UNIT_02.CYCLE_SELECTED_AUX) AND (("DB2440_GLOBAL_DATA".GLOBAL_DATA.U02_RN_CYCLE_PART_TYPE AND (("DB2031_CYCLES_GENERAL".MANUAL_LOAD_CYCLE.CYCLE_SELECTED AND "DB8100_MANUAL_LOADING_PART_STATUS".UNIT_02_NO_FACE_R_PARTS_TO_DELIVER) OR (NOT "DB2031_CYCLES_GENERAL".MANUAL_LOAD_CYCLE.CYCLE_SELECTED AND NOT "DB7330_ETXETAR_ROBOT_CELL_INTERLOCK".INTERLOCKS_UNIT_02.ROBOT_TO_MACHINE.RBT_PART_FACE_R_TO_DELIVER)) AND ("DB4000_FIX_TABLE_POSITIONS".UNIT_02.FIXTURE_1.IN_LOAD_UNLOAD_STATION_1 OR "DB4000_FIX_TABLE_POSITIONS".UNIT_02.FIXTURE_3.IN_LOAD_UNLOAD_STATION_1 OR ((("DB2031_CYCLES_GENERAL".MANUAL_LOAD_CYCLE.CYCLE_SELECTED AND (("DB8100_MANUAL_LOADING_PART_STATUS".UNIT_02_NO_FACE_N_PARTS_TO_DELIVER AND NOT "DB8101_MANUAL_LOADING_PART_STATUS_MANAGEMENT".UNIT_02_INTERMEDIATE.STATUS.PRESENT) OR "DB2440_GLOBAL_DATA".GLOBAL_DATA.UNIT_02_PART_PRESENT)) OR (NOT "DB2031_CYCLES_GENERAL".MANUAL_LOAD_CYCLE.CYCLE_SELECTED AND ((NOT "DB7330_ETXETAR_ROBOT_CELL_INTERLOCK".INTERLOCKS_UNIT_02.ROBOT_TO_MACHINE.RBT_PART_FACE_N_TO_DELIVER AND NOT "DB8101_MANUAL_LOADING_PART_STATUS_MANAGEMENT".UNIT_02_INTERMEDIATE.STATUS.PRESENT) OR "DB2440_GLOBAL_DATA".GLOBAL_DATA.UNIT_02_PART_PRESENT))) AND ("DB4000_FIX_TABLE_POSITIONS".UNIT_02.FIXTURE_2.IN_LOAD_UNLOAD_STATION_1 OR "DB4000_FIX_TABLE_POSITIONS".UNIT_02.FIXTURE_4.IN_LOAD_UNLOAD_STATION_1)))) OR ("DB2440_GLOBAL_DATA".GLOBAL_DATA.U02_NR_CYCLE_PART_TYPE AND (("DB2031_CYCLES_GENERAL".MANUAL_LOAD_CYCLE.CYCLE_SELECTED AND "DB8100_MANUAL_LOADING_PART_STATUS".UNIT_02_NO_FACE_N_PARTS_TO_DELIVER) OR (NOT "DB2031_CYCLES_GENERAL".MANUAL_LOAD_CYCLE.CYCLE_SELECTED AND NOT "DB7330_ETXETAR_ROBOT_CELL_INTERLOCK".INTERLOCKS_UNIT_02.ROBOT_TO_MACHINE.RBT_PART_FACE_N_TO_DELIVER)) AND ("DB4000_FIX_TABLE_POSITIONS".UNIT_02.FIXTURE_2.IN_LOAD_UNLOAD_STATION_1 OR "DB4000_FIX_TABLE_POSITIONS".UNIT_02.FIXTURE_4.IN_LOAD_UNLOAD_STATION_1 OR ((("DB2031_CYCLES_GENERAL".MANUAL_LOAD_CYCLE.CYCLE_SELECTED AND (("DB8100_MANUAL_LOADING_PART_STATUS".UNIT_02_NO_FACE_R_PARTS_TO_DELIVER AND NOT "DB8101_MANUAL_LOADING_PART_STATUS_MANAGEMENT".UNIT_02_INTERMEDIATE.STATUS.PRESENT) OR "DB2440_GLOBAL_DATA".GLOBAL_DATA.UNIT_02_PART_PRESENT)) OR (NOT "DB2031_CYCLES_GENERAL".MANUAL_LOAD_CYCLE.CYCLE_SELECTED AND (NOT "DB7330_ETXETAR_ROBOT_CELL_INTERLOCK".INTERLOCKS_UNIT_02.ROBOT_TO_MACHINE.RBT_PART_FACE_R_TO_DELIVER OR "DB2440_GLOBAL_DATA".GLOBAL_DATA.UNIT_02_PART_PRESENT))) AND ("DB4000_FIX_TABLE_POSITIONS".UNIT_02.FIXTURE_1.IN_LOAD_UNLOAD_STATION_1 OR "DB4000_FIX_TABLE_POSITIONS".UNIT_02.FIXTURE_3.IN_LOAD_UNLOAD_STATION_1)))))))) OR ("DB1101_MACHINE_SEQUENCE".SKIP_FIXTURE_UNIT_02 AND NOT "DB4000_FIX_TABLE_POSITIONS".UNIT_02.AXIS_E20_NOT_DEFINED_POS AND "DB1251_PART_CYCLE_UNIT_02".RUNNING);
END_REGION

REGION Network 16: CYCLE UNIT 01
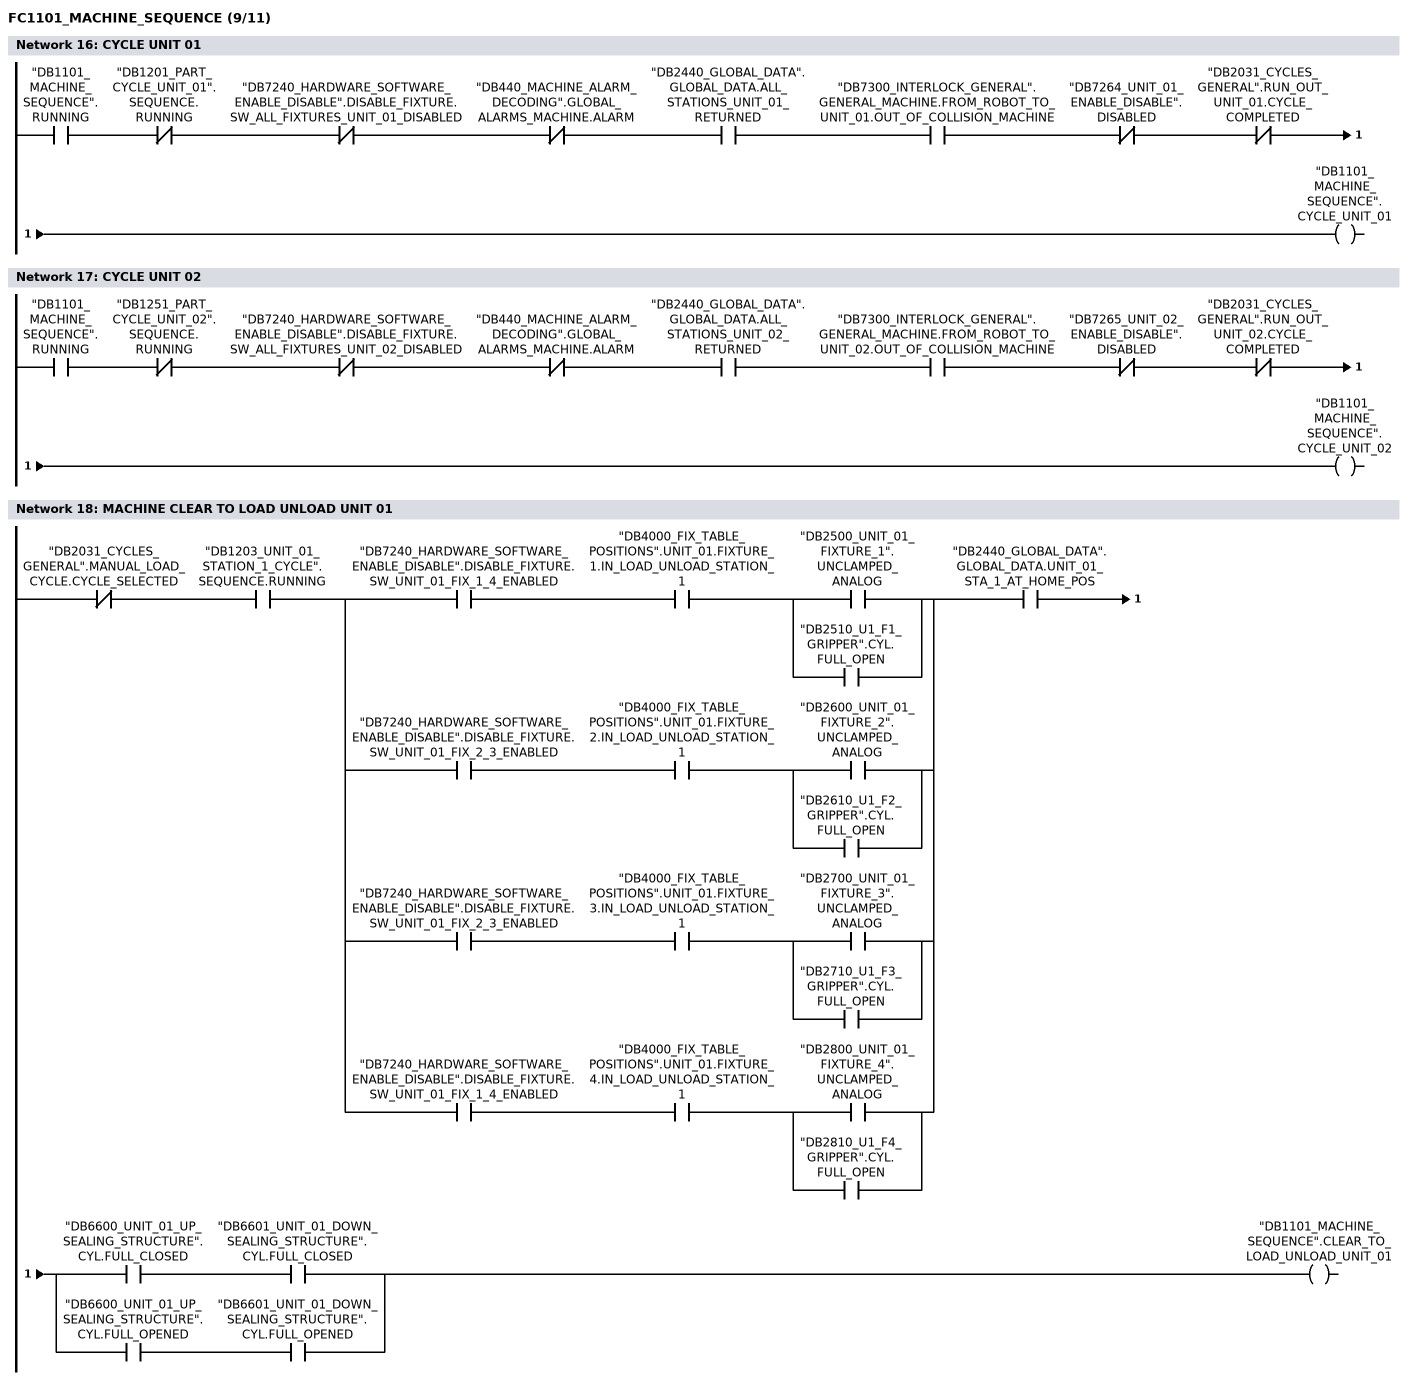
   RUNG wire#powerrail
      Contact( "DB1101_MACHINE_SEQUENCE".RUNNING )
      I_Contact( "DB1201_PART_CYCLE_UNIT_01".SEQUENCE.RUNNING )
      I_Contact( "DB7240_HARDWARE_SOFTWARE_ENABLE_DISABLE".DISABLE_FIXTURE.SW_ALL_FIXTURES_UNIT_01_DISABLED )
      I_Contact( "DB440_MACHINE_ALARM_DECODING".GLOBAL_ALARMS_MACHINE.ALARM )
      Contact( "DB2440_GLOBAL_DATA".GLOBAL_DATA.ALL_STATIONS_UNIT_01_RETURNED )
      Contact( "DB7300_INTERLOCK_GENERAL".GENERAL_MACHINE.FROM_ROBOT_TO_UNIT_01.OUT_OF_COLLISION_MACHINE )
      I_Contact( "DB7264_UNIT_01_ENABLE_DISABLE".DISABLED )
      I_Contact( "DB2031_CYCLES_GENERAL".RUN_OUT_UNIT_01.CYCLE_COMPLETED )
      Coil( "DB1101_MACHINE_SEQUENCE".CYCLE_UNIT_01 )
   END_RUNG
   // the same network as SCL:
   "DB1101_MACHINE_SEQUENCE".CYCLE_UNIT_01 := "DB1101_MACHINE_SEQUENCE".RUNNING AND NOT "DB1201_PART_CYCLE_UNIT_01".SEQUENCE.RUNNING AND NOT "DB7240_HARDWARE_SOFTWARE_ENABLE_DISABLE".DISABLE_FIXTURE.SW_ALL_FIXTURES_UNIT_01_DISABLED AND NOT "DB440_MACHINE_ALARM_DECODING".GLOBAL_ALARMS_MACHINE.ALARM AND "DB2440_GLOBAL_DATA".GLOBAL_DATA.ALL_STATIONS_UNIT_01_RETURNED AND "DB7300_INTERLOCK_GENERAL".GENERAL_MACHINE.FROM_ROBOT_TO_UNIT_01.OUT_OF_COLLISION_MACHINE AND NOT "DB7264_UNIT_01_ENABLE_DISABLE".DISABLED AND NOT "DB2031_CYCLES_GENERAL".RUN_OUT_UNIT_01.CYCLE_COMPLETED;
END_REGION

REGION Network 17: CYCLE UNIT 02
   RUNG wire#powerrail
      Contact( "DB1101_MACHINE_SEQUENCE".RUNNING )
      I_Contact( "DB1251_PART_CYCLE_UNIT_02".SEQUENCE.RUNNING )
      I_Contact( "DB7240_HARDWARE_SOFTWARE_ENABLE_DISABLE".DISABLE_FIXTURE.SW_ALL_FIXTURES_UNIT_02_DISABLED )
      I_Contact( "DB440_MACHINE_ALARM_DECODING".GLOBAL_ALARMS_MACHINE.ALARM )
      Contact( "DB2440_GLOBAL_DATA".GLOBAL_DATA.ALL_STATIONS_UNIT_02_RETURNED )
      Contact( "DB7300_INTERLOCK_GENERAL".GENERAL_MACHINE.FROM_ROBOT_TO_UNIT_02.OUT_OF_COLLISION_MACHINE )
      I_Contact( "DB7265_UNIT_02_ENABLE_DISABLE".DISABLED )
      I_Contact( "DB2031_CYCLES_GENERAL".RUN_OUT_UNIT_02.CYCLE_COMPLETED )
      Coil( "DB1101_MACHINE_SEQUENCE".CYCLE_UNIT_02 )
   END_RUNG
   // the same network as SCL:
   "DB1101_MACHINE_SEQUENCE".CYCLE_UNIT_02 := "DB1101_MACHINE_SEQUENCE".RUNNING AND NOT "DB1251_PART_CYCLE_UNIT_02".SEQUENCE.RUNNING AND NOT "DB7240_HARDWARE_SOFTWARE_ENABLE_DISABLE".DISABLE_FIXTURE.SW_ALL_FIXTURES_UNIT_02_DISABLED AND NOT "DB440_MACHINE_ALARM_DECODING".GLOBAL_ALARMS_MACHINE.ALARM AND "DB2440_GLOBAL_DATA".GLOBAL_DATA.ALL_STATIONS_UNIT_02_RETURNED AND "DB7300_INTERLOCK_GENERAL".GENERAL_MACHINE.FROM_ROBOT_TO_UNIT_02.OUT_OF_COLLISION_MACHINE AND NOT "DB7265_UNIT_02_ENABLE_DISABLE".DISABLED AND NOT "DB2031_CYCLES_GENERAL".RUN_OUT_UNIT_02.CYCLE_COMPLETED;
END_REGION

REGION Network 18: MACHINE CLEAR TO LOAD UNLOAD UNIT 01
   RUNG wire#powerrail
      I_Contact( "DB2031_CYCLES_GENERAL".MANUAL_LOAD_CYCLE.CYCLE_SELECTED )
      Contact( "DB1203_UNIT_01_STATION_1_CYCLE".SEQUENCE.RUNNING )
      wire#w1
      Contact( "DB7240_HARDWARE_SOFTWARE_ENABLE_DISABLE".DISABLE_FIXTURE.SW_UNIT_01_FIX_1_4_ENABLED )
      Contact( "DB4000_FIX_TABLE_POSITIONS".UNIT_01.FIXTURE_1.IN_LOAD_UNLOAD_STATION_1 )
      wire#w2
      Contact( "DB2500_UNIT_01_FIXTURE_1".UNCLAMPED_ANALOG )
      wire#w3
      Contact( "DB2440_GLOBAL_DATA".GLOBAL_DATA.UNIT_01_STA_1_AT_HOME_POS )
      wire#w7
      Contact( "DB6600_UNIT_01_UP_SEALING_STRUCTURE".CYL.FULL_CLOSED )
      Contact( "DB6601_UNIT_01_DOWN_SEALING_STRUCTURE".CYL.FULL_CLOSED )
      wire#w8
      Coil( "DB1101_MACHINE_SEQUENCE".CLEAR_TO_LOAD_UNLOAD_UNIT_01 )
   END_RUNG
   RUNG wire#w2
      Contact( "DB2510_U1_F1_GRIPPER".CYL.FULL_OPEN )
   END_RUNG wire#w3
   RUNG wire#w1
      Contact( "DB7240_HARDWARE_SOFTWARE_ENABLE_DISABLE".DISABLE_FIXTURE.SW_UNIT_01_FIX_2_3_ENABLED )
      Contact( "DB4000_FIX_TABLE_POSITIONS".UNIT_01.FIXTURE_2.IN_LOAD_UNLOAD_STATION_1 )
      wire#w4
      Contact( "DB2600_UNIT_01_FIXTURE_2".UNCLAMPED_ANALOG )
   END_RUNG wire#w3
   RUNG wire#w4
      Contact( "DB2610_U1_F2_GRIPPER".CYL.FULL_OPEN )
   END_RUNG wire#w3
   RUNG wire#w1
      Contact( "DB7240_HARDWARE_SOFTWARE_ENABLE_DISABLE".DISABLE_FIXTURE.SW_UNIT_01_FIX_2_3_ENABLED )
      Contact( "DB4000_FIX_TABLE_POSITIONS".UNIT_01.FIXTURE_3.IN_LOAD_UNLOAD_STATION_1 )
      wire#w5
      Contact( "DB2700_UNIT_01_FIXTURE_3".UNCLAMPED_ANALOG )
   END_RUNG wire#w3
   RUNG wire#w5
      Contact( "DB2710_U1_F3_GRIPPER".CYL.FULL_OPEN )
   END_RUNG wire#w3
   RUNG wire#w1
      Contact( "DB7240_HARDWARE_SOFTWARE_ENABLE_DISABLE".DISABLE_FIXTURE.SW_UNIT_01_FIX_1_4_ENABLED )
      Contact( "DB4000_FIX_TABLE_POSITIONS".UNIT_01.FIXTURE_4.IN_LOAD_UNLOAD_STATION_1 )
      wire#w6
      Contact( "DB2800_UNIT_01_FIXTURE_4".UNCLAMPED_ANALOG )
   END_RUNG wire#w3
   RUNG wire#w6
      Contact( "DB2810_U1_F4_GRIPPER".CYL.FULL_OPEN )
   END_RUNG wire#w3
   RUNG wire#w7
      Contact( "DB6600_UNIT_01_UP_SEALING_STRUCTURE".CYL.FULL_OPENED )
      Contact( "DB6601_UNIT_01_DOWN_SEALING_STRUCTURE".CYL.FULL_OPENED )
   END_RUNG wire#w8
   // the same network as SCL:
   "DB1101_MACHINE_SEQUENCE".CLEAR_TO_LOAD_UNLOAD_UNIT_01 := NOT "DB2031_CYCLES_GENERAL".MANUAL_LOAD_CYCLE.CYCLE_SELECTED AND "DB1203_UNIT_01_STATION_1_CYCLE".SEQUENCE.RUNNING AND (("DB7240_HARDWARE_SOFTWARE_ENABLE_DISABLE".DISABLE_FIXTURE.SW_UNIT_01_FIX_1_4_ENABLED AND "DB4000_FIX_TABLE_POSITIONS".UNIT_01.FIXTURE_1.IN_LOAD_UNLOAD_STATION_1 AND ("DB2500_UNIT_01_FIXTURE_1".UNCLAMPED_ANALOG OR "DB2510_U1_F1_GRIPPER".CYL.FULL_OPEN)) OR ("DB7240_HARDWARE_SOFTWARE_ENABLE_DISABLE".DISABLE_FIXTURE.SW_UNIT_01_FIX_2_3_ENABLED AND "DB4000_FIX_TABLE_POSITIONS".UNIT_01.FIXTURE_2.IN_LOAD_UNLOAD_STATION_1 AND ("DB2600_UNIT_01_FIXTURE_2".UNCLAMPED_ANALOG OR "DB2610_U1_F2_GRIPPER".CYL.FULL_OPEN)) OR ("DB7240_HARDWARE_SOFTWARE_ENABLE_DISABLE".DISABLE_FIXTURE.SW_UNIT_01_FIX_2_3_ENABLED AND "DB4000_FIX_TABLE_POSITIONS".UNIT_01.FIXTURE_3.IN_LOAD_UNLOAD_STATION_1 AND ("DB2700_UNIT_01_FIXTURE_3".UNCLAMPED_ANALOG OR "DB2710_U1_F3_GRIPPER".CYL.FULL_OPEN)) OR ("DB7240_HARDWARE_SOFTWARE_ENABLE_DISABLE".DISABLE_FIXTURE.SW_UNIT_01_FIX_1_4_ENABLED AND "DB4000_FIX_TABLE_POSITIONS".UNIT_01.FIXTURE_4.IN_LOAD_UNLOAD_STATION_1 AND ("DB2800_UNIT_01_FIXTURE_4".UNCLAMPED_ANALOG OR "DB2810_U1_F4_GRIPPER".CYL.FULL_OPEN))) AND "DB2440_GLOBAL_DATA".GLOBAL_DATA.UNIT_01_STA_1_AT_HOME_POS AND (("DB6600_UNIT_01_UP_SEALING_STRUCTURE".CYL.FULL_CLOSED AND "DB6601_UNIT_01_DOWN_SEALING_STRUCTURE".CYL.FULL_CLOSED) OR ("DB6600_UNIT_01_UP_SEALING_STRUCTURE".CYL.FULL_OPENED AND "DB6601_UNIT_01_DOWN_SEALING_STRUCTURE".CYL.FULL_OPENED));
END_REGION

REGION Network 19: MACHINE CLEAR TO LOAD UNLOAD UNIT 02
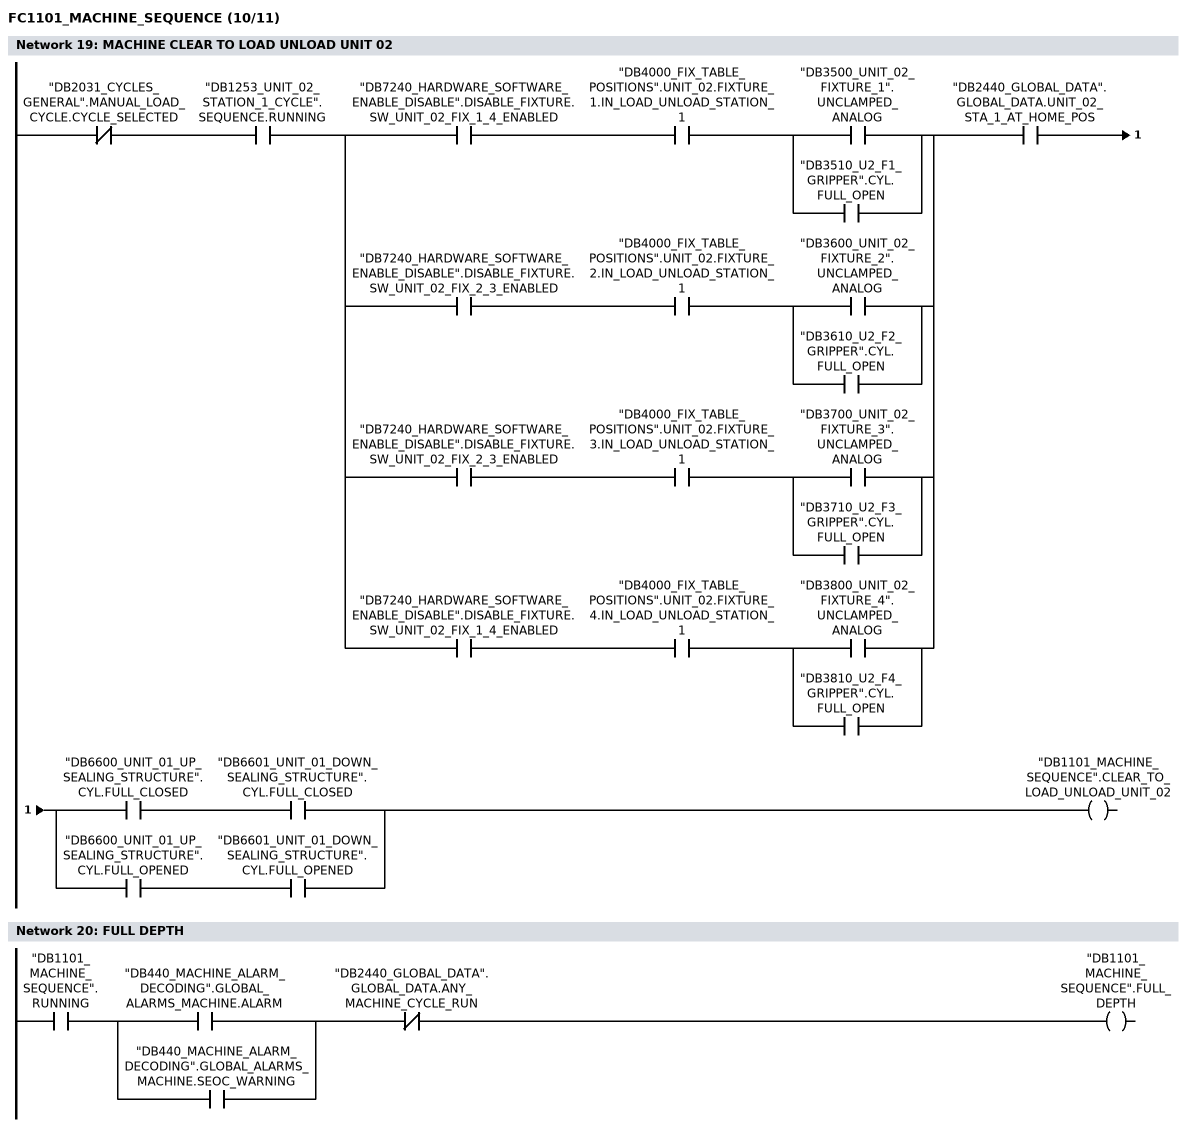
   RUNG wire#powerrail
      I_Contact( "DB2031_CYCLES_GENERAL".MANUAL_LOAD_CYCLE.CYCLE_SELECTED )
      Contact( "DB1253_UNIT_02_STATION_1_CYCLE".SEQUENCE.RUNNING )
      wire#w1
      Contact( "DB7240_HARDWARE_SOFTWARE_ENABLE_DISABLE".DISABLE_FIXTURE.SW_UNIT_02_FIX_1_4_ENABLED )
      Contact( "DB4000_FIX_TABLE_POSITIONS".UNIT_02.FIXTURE_1.IN_LOAD_UNLOAD_STATION_1 )
      wire#w2
      Contact( "DB3500_UNIT_02_FIXTURE_1".UNCLAMPED_ANALOG )
      wire#w3
      Contact( "DB2440_GLOBAL_DATA".GLOBAL_DATA.UNIT_02_STA_1_AT_HOME_POS )
      wire#w7
      Contact( "DB6600_UNIT_01_UP_SEALING_STRUCTURE".CYL.FULL_CLOSED )
      Contact( "DB6601_UNIT_01_DOWN_SEALING_STRUCTURE".CYL.FULL_CLOSED )
      wire#w8
      Coil( "DB1101_MACHINE_SEQUENCE".CLEAR_TO_LOAD_UNLOAD_UNIT_02 )
   END_RUNG
   RUNG wire#w2
      Contact( "DB3510_U2_F1_GRIPPER".CYL.FULL_OPEN )
   END_RUNG wire#w3
   RUNG wire#w1
      Contact( "DB7240_HARDWARE_SOFTWARE_ENABLE_DISABLE".DISABLE_FIXTURE.SW_UNIT_02_FIX_2_3_ENABLED )
      Contact( "DB4000_FIX_TABLE_POSITIONS".UNIT_02.FIXTURE_2.IN_LOAD_UNLOAD_STATION_1 )
      wire#w4
      Contact( "DB3600_UNIT_02_FIXTURE_2".UNCLAMPED_ANALOG )
   END_RUNG wire#w3
   RUNG wire#w4
      Contact( "DB3610_U2_F2_GRIPPER".CYL.FULL_OPEN )
   END_RUNG wire#w3
   RUNG wire#w1
      Contact( "DB7240_HARDWARE_SOFTWARE_ENABLE_DISABLE".DISABLE_FIXTURE.SW_UNIT_02_FIX_2_3_ENABLED )
      Contact( "DB4000_FIX_TABLE_POSITIONS".UNIT_02.FIXTURE_3.IN_LOAD_UNLOAD_STATION_1 )
      wire#w5
      Contact( "DB3700_UNIT_02_FIXTURE_3".UNCLAMPED_ANALOG )
   END_RUNG wire#w3
   RUNG wire#w5
      Contact( "DB3710_U2_F3_GRIPPER".CYL.FULL_OPEN )
   END_RUNG wire#w3
   RUNG wire#w1
      Contact( "DB7240_HARDWARE_SOFTWARE_ENABLE_DISABLE".DISABLE_FIXTURE.SW_UNIT_02_FIX_1_4_ENABLED )
      Contact( "DB4000_FIX_TABLE_POSITIONS".UNIT_02.FIXTURE_4.IN_LOAD_UNLOAD_STATION_1 )
      wire#w6
      Contact( "DB3800_UNIT_02_FIXTURE_4".UNCLAMPED_ANALOG )
   END_RUNG wire#w3
   RUNG wire#w6
      Contact( "DB3810_U2_F4_GRIPPER".CYL.FULL_OPEN )
   END_RUNG wire#w3
   RUNG wire#w7
      Contact( "DB6600_UNIT_01_UP_SEALING_STRUCTURE".CYL.FULL_OPENED )
      Contact( "DB6601_UNIT_01_DOWN_SEALING_STRUCTURE".CYL.FULL_OPENED )
   END_RUNG wire#w8
   // the same network as SCL:
   "DB1101_MACHINE_SEQUENCE".CLEAR_TO_LOAD_UNLOAD_UNIT_02 := NOT "DB2031_CYCLES_GENERAL".MANUAL_LOAD_CYCLE.CYCLE_SELECTED AND "DB1253_UNIT_02_STATION_1_CYCLE".SEQUENCE.RUNNING AND (("DB7240_HARDWARE_SOFTWARE_ENABLE_DISABLE".DISABLE_FIXTURE.SW_UNIT_02_FIX_1_4_ENABLED AND "DB4000_FIX_TABLE_POSITIONS".UNIT_02.FIXTURE_1.IN_LOAD_UNLOAD_STATION_1 AND ("DB3500_UNIT_02_FIXTURE_1".UNCLAMPED_ANALOG OR "DB3510_U2_F1_GRIPPER".CYL.FULL_OPEN)) OR ("DB7240_HARDWARE_SOFTWARE_ENABLE_DISABLE".DISABLE_FIXTURE.SW_UNIT_02_FIX_2_3_ENABLED AND "DB4000_FIX_TABLE_POSITIONS".UNIT_02.FIXTURE_2.IN_LOAD_UNLOAD_STATION_1 AND ("DB3600_UNIT_02_FIXTURE_2".UNCLAMPED_ANALOG OR "DB3610_U2_F2_GRIPPER".CYL.FULL_OPEN)) OR ("DB7240_HARDWARE_SOFTWARE_ENABLE_DISABLE".DISABLE_FIXTURE.SW_UNIT_02_FIX_2_3_ENABLED AND "DB4000_FIX_TABLE_POSITIONS".UNIT_02.FIXTURE_3.IN_LOAD_UNLOAD_STATION_1 AND ("DB3700_UNIT_02_FIXTURE_3".UNCLAMPED_ANALOG OR "DB3710_U2_F3_GRIPPER".CYL.FULL_OPEN)) OR ("DB7240_HARDWARE_SOFTWARE_ENABLE_DISABLE".DISABLE_FIXTURE.SW_UNIT_02_FIX_1_4_ENABLED AND "DB4000_FIX_TABLE_POSITIONS".UNIT_02.FIXTURE_4.IN_LOAD_UNLOAD_STATION_1 AND ("DB3800_UNIT_02_FIXTURE_4".UNCLAMPED_ANALOG OR "DB3810_U2_F4_GRIPPER".CYL.FULL_OPEN))) AND "DB2440_GLOBAL_DATA".GLOBAL_DATA.UNIT_02_STA_1_AT_HOME_POS AND (("DB6600_UNIT_01_UP_SEALING_STRUCTURE".CYL.FULL_CLOSED AND "DB6601_UNIT_01_DOWN_SEALING_STRUCTURE".CYL.FULL_CLOSED) OR ("DB6600_UNIT_01_UP_SEALING_STRUCTURE".CYL.FULL_OPENED AND "DB6601_UNIT_01_DOWN_SEALING_STRUCTURE".CYL.FULL_OPENED));
END_REGION

REGION Network 20: FULL DEPTH
   RUNG wire#powerrail
      Contact( "DB1101_MACHINE_SEQUENCE".RUNNING )
      wire#w1
      Contact( "DB440_MACHINE_ALARM_DECODING".GLOBAL_ALARMS_MACHINE.ALARM )
      wire#w2
      I_Contact( "DB2440_GLOBAL_DATA".GLOBAL_DATA.ANY_MACHINE_CYCLE_RUN )
      Coil( "DB1101_MACHINE_SEQUENCE".FULL_DEPTH )
   END_RUNG
   RUNG wire#w1
      Contact( "DB440_MACHINE_ALARM_DECODING".GLOBAL_ALARMS_MACHINE.SEOC_WARNING )
   END_RUNG wire#w2
   // the same network as SCL:
   "DB1101_MACHINE_SEQUENCE".FULL_DEPTH := "DB1101_MACHINE_SEQUENCE".RUNNING AND ("DB440_MACHINE_ALARM_DECODING".GLOBAL_ALARMS_MACHINE.ALARM OR "DB440_MACHINE_ALARM_DECODING".GLOBAL_ALARMS_MACHINE.SEOC_WARNING) AND NOT "DB2440_GLOBAL_DATA".GLOBAL_DATA.ANY_MACHINE_CYCLE_RUN;
END_REGION

REGION Network 21: TIME EXCEEDED ALARM
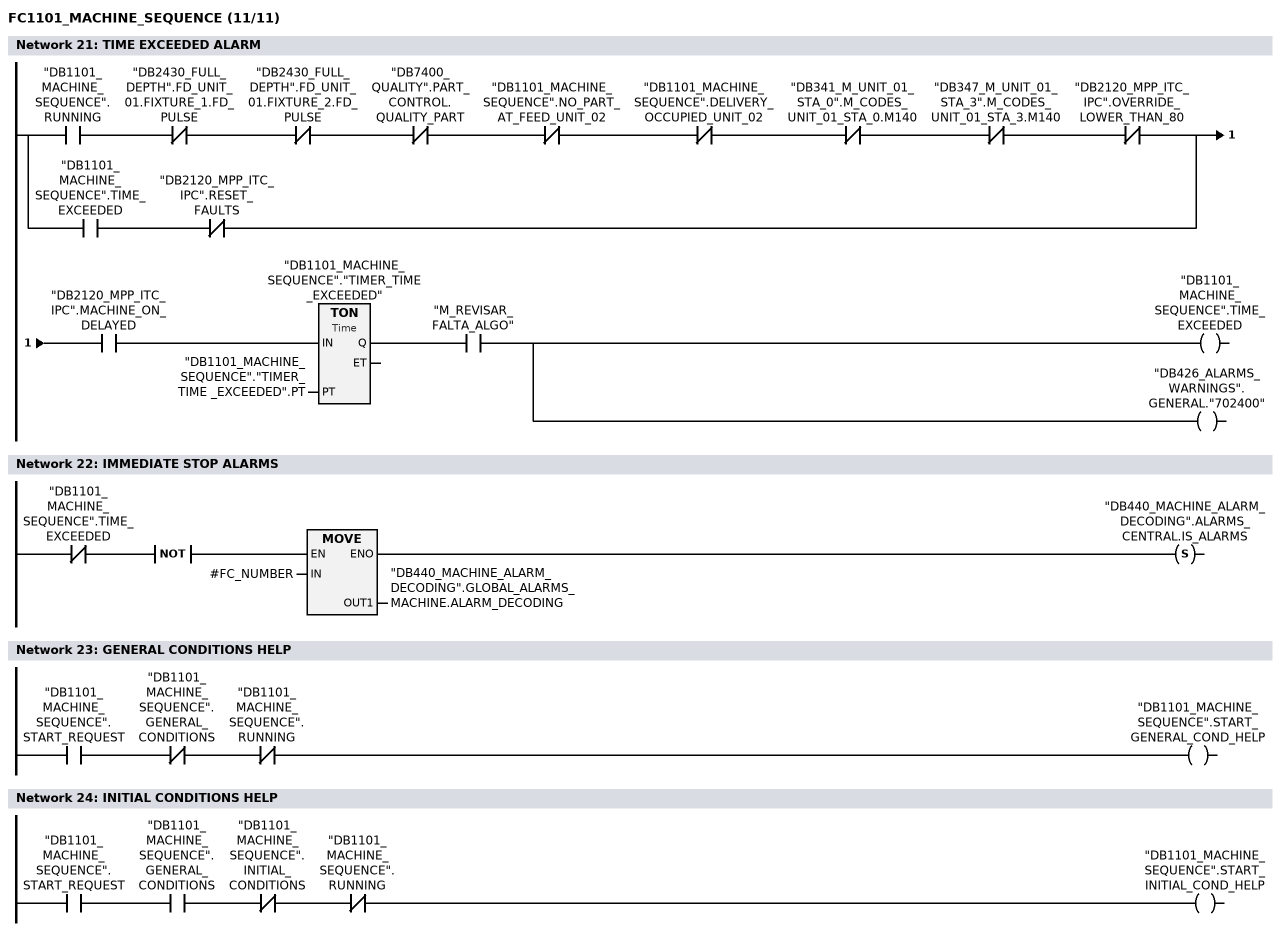
   RUNG wire#powerrail
      Contact( "DB1101_MACHINE_SEQUENCE".RUNNING )
      I_Contact( "DB2430_FULL_DEPTH".FD_UNIT_01.FIXTURE_1.FD_PULSE )
      I_Contact( "DB2430_FULL_DEPTH".FD_UNIT_01.FIXTURE_2.FD_PULSE )
      I_Contact( "DB7400_QUALITY".PART_CONTROL.QUALITY_PART )
      I_Contact( "DB1101_MACHINE_SEQUENCE".NO_PART_AT_FEED_UNIT_02 )
      I_Contact( "DB1101_MACHINE_SEQUENCE".DELIVERY_OCCUPIED_UNIT_02 )
      I_Contact( "DB341_M_UNIT_01_STA_0".M_CODES_UNIT_01_STA_0.M140 )
      I_Contact( "DB347_M_UNIT_01_STA_3".M_CODES_UNIT_01_STA_3.M140 )
      I_Contact( "DB2120_MPP_ITC_IPC".OVERRIDE_LOWER_THAN_80 )
      wire#w1
      Contact( "DB2120_MPP_ITC_IPC".MACHINE_ON_DELAYED )
      { S7_Templates := "time_type := Time" } "DB1101_MACHINE_SEQUENCE"."TIMER_TIME _EXCEEDED".TON(pt := "DB1101_MACHINE_SEQUENCE"."TIMER_TIME _EXCEEDED".PT, et =>)
      Contact( "M_REVISAR_FALTA_ALGO" )
      wire#w2
      Coil( "DB1101_MACHINE_SEQUENCE".TIME_EXCEEDED )
   END_RUNG
   RUNG wire#powerrail
      Contact( "DB1101_MACHINE_SEQUENCE".TIME_EXCEEDED )
      I_Contact( "DB2120_MPP_ITC_IPC".RESET_FAULTS )
   END_RUNG wire#w1
   RUNG wire#w2
      Coil( "DB426_ALARMS_WARNINGS".GENERAL."702400" )
   END_RUNG
   // the same network as SCL:
   "DB1101_MACHINE_SEQUENCE"."TIMER_TIME _EXCEEDED".TON(IN := (("DB1101_MACHINE_SEQUENCE".RUNNING AND NOT "DB2430_FULL_DEPTH".FD_UNIT_01.FIXTURE_1.FD_PULSE AND NOT "DB2430_FULL_DEPTH".FD_UNIT_01.FIXTURE_2.FD_PULSE AND NOT "DB7400_QUALITY".PART_CONTROL.QUALITY_PART AND NOT "DB1101_MACHINE_SEQUENCE".NO_PART_AT_FEED_UNIT_02 AND NOT "DB1101_MACHINE_SEQUENCE".DELIVERY_OCCUPIED_UNIT_02 AND NOT "DB341_M_UNIT_01_STA_0".M_CODES_UNIT_01_STA_0.M140 AND NOT "DB347_M_UNIT_01_STA_3".M_CODES_UNIT_01_STA_3.M140 AND NOT "DB2120_MPP_ITC_IPC".OVERRIDE_LOWER_THAN_80) OR ("DB1101_MACHINE_SEQUENCE".TIME_EXCEEDED AND NOT "DB2120_MPP_ITC_IPC".RESET_FAULTS)) AND "DB2120_MPP_ITC_IPC".MACHINE_ON_DELAYED,
                           PT := "DB1101_MACHINE_SEQUENCE"."TIMER_TIME _EXCEEDED".PT);
   "DB1101_MACHINE_SEQUENCE".TIME_EXCEEDED := "DB1101_MACHINE_SEQUENCE"."TIMER_TIME _EXCEEDED".Q AND "M_REVISAR_FALTA_ALGO";
   "DB426_ALARMS_WARNINGS".GENERAL."702400" := "DB1101_MACHINE_SEQUENCE".TIME_EXCEEDED;
END_REGION

REGION Network 22: IMMEDIATE STOP ALARMS
   RUNG wire#powerrail
      I_Contact( "DB1101_MACHINE_SEQUENCE".TIME_EXCEEDED )
      Not()
      { S7_GenerateENO := "TRUE" } Move(in := #FC_NUMBER, out1 => "DB440_MACHINE_ALARM_DECODING".GLOBAL_ALARMS_MACHINE.ALARM_DECODING)
      S_Coil( "DB440_MACHINE_ALARM_DECODING".ALARMS_CENTRAL.IS_ALARMS )
   END_RUNG
   // the same network as SCL:
   // ENO of a box is taken as its EN; it also drops when the box reports an error
   IF NOT (NOT "DB1101_MACHINE_SEQUENCE".TIME_EXCEEDED) THEN
       "DB440_MACHINE_ALARM_DECODING".GLOBAL_ALARMS_MACHINE.ALARM_DECODING := #FC_NUMBER;
       "DB440_MACHINE_ALARM_DECODING".ALARMS_CENTRAL.IS_ALARMS := TRUE;
   END_IF;
END_REGION

REGION Network 23: GENERAL CONDITIONS HELP
   RUNG wire#powerrail
      Contact( "DB1101_MACHINE_SEQUENCE".START_REQUEST )
      I_Contact( "DB1101_MACHINE_SEQUENCE".GENERAL_CONDITIONS )
      I_Contact( "DB1101_MACHINE_SEQUENCE".RUNNING )
      Coil( "DB1101_MACHINE_SEQUENCE".START_GENERAL_COND_HELP )
   END_RUNG
   // the same network as SCL:
   "DB1101_MACHINE_SEQUENCE".START_GENERAL_COND_HELP := "DB1101_MACHINE_SEQUENCE".START_REQUEST AND NOT "DB1101_MACHINE_SEQUENCE".GENERAL_CONDITIONS AND NOT "DB1101_MACHINE_SEQUENCE".RUNNING;
END_REGION

REGION Network 24: INITIAL CONDITIONS HELP
   RUNG wire#powerrail
      Contact( "DB1101_MACHINE_SEQUENCE".START_REQUEST )
      Contact( "DB1101_MACHINE_SEQUENCE".GENERAL_CONDITIONS )
      I_Contact( "DB1101_MACHINE_SEQUENCE".INITIAL_CONDITIONS )
      I_Contact( "DB1101_MACHINE_SEQUENCE".RUNNING )
      Coil( "DB1101_MACHINE_SEQUENCE".START_INITIAL_COND_HELP )
   END_RUNG
   // the same network as SCL:
   "DB1101_MACHINE_SEQUENCE".START_INITIAL_COND_HELP := "DB1101_MACHINE_SEQUENCE".START_REQUEST AND "DB1101_MACHINE_SEQUENCE".GENERAL_CONDITIONS AND NOT "DB1101_MACHINE_SEQUENCE".INITIAL_CONDITIONS AND NOT "DB1101_MACHINE_SEQUENCE".RUNNING;
END_REGION
END_FUNCTION
